    movel([0.209810, -1.227135, -2.664423, -0.820831, 1.570796, 1.780606],accel_mss,speed_ms,0,blend_radius_m)
    movel([0.209627, -1.226934, -2.664525, -0.820930, 1.570796, 1.780424],accel_mss,speed_ms,0,blend_radius_m)
    movel([0.208422, -1.226483, -2.664753, -0.821153, 1.570796, 1.779219],accel_mss,speed_ms,0,blend_radius_m)
    movel([0.205590, -1.225749, -2.665124, -0.821516, 1.570796, 1.776387],accel_mss,speed_ms,0,blend_radius_m)
    movel([0.202937, -1.225278, -2.665361, -0.821749, 1.570796, 1.773733],accel_mss,speed_ms,0,blend_radius_m)
    movel([0.200496, -1.225073, -2.665465, -0.821852, 1.570796, 1.771292],accel_mss,speed_ms,0,blend_radius_m)
    movel([0.198313, -1.225138, -2.665432, -0.821819, 1.570796, 1.769109],accel_mss,speed_ms,0,blend_radius_m)
    movel([0.196815, -1.225270, -2.665365, -0.821754, 1.570796, 1.767612],accel_mss,speed_ms,0,blend_radius_m)
    movel([0.196665, -1.225161, -2.665420, -0.821808, 1.570796, 1.767461],accel_mss,speed_ms,0,blend_radius_m)
    movel([0.196789, -1.224942, -2.665530, -0.821916, 1.570796, 1.767585],accel_mss,speed_ms,0,blend_radius_m)
    movel([0.198166, -1.223979, -2.666015, -0.822395, 1.570796, 1.768963],accel_mss,speed_ms,0,blend_radius_m)
    movel([0.198894, -1.223467, -2.666272, -0.822649, 1.570796, 1.769690],accel_mss,speed_ms,0,blend_radius_m)
    movel([0.200219, -1.222435, -2.666790, -0.823164, 1.570796, 1.771015],accel_mss,speed_ms,0,blend_radius_m)
    movel([0.200325, -1.222080, -2.666968, -0.823342, 1.570796, 1.771122],accel_mss,speed_ms,0,blend_radius_m)
    movel([0.200128, -1.221809, -2.667103, -0.823477, 1.570796, 1.770925],accel_mss,speed_ms,0,blend_radius_m)
    movel([0.199567, -1.221632, -2.667191, -0.823565, 1.570796, 1.770363],accel_mss,speed_ms,0,blend_radius_m)
    movel([0.198593, -1.221552, -2.667232, -0.823605, 1.570796, 1.769390],accel_mss,speed_ms,0,blend_radius_m)
    movel([0.196633, -1.221578, -2.667219, -0.823592, 1.570796, 1.767430],accel_mss,speed_ms,0,blend_radius_m)
    movel([0.194680, -1.221799, -2.667108, -0.823482, 1.570796, 1.765476],accel_mss,speed_ms,0,blend_radius_m)
    movel([0.192596, -1.222232, -2.666892, -0.823266, 1.570796, 1.763392],accel_mss,speed_ms,0,blend_radius_m)
    movel([0.187306, -1.223836, -2.666087, -0.822466, 1.570796, 1.758102],accel_mss,speed_ms,0,blend_radius_m)
    movel([0.188189, -1.223147, -2.666433, -0.822809, 1.570796, 1.758986],accel_mss,speed_ms,0,blend_radius_m)
    movel([0.190951, -1.221398, -2.667309, -0.823682, 1.570796, 1.761748],accel_mss,speed_ms,0,blend_radius_m)
    movel([0.191998, -1.220793, -2.667611, -0.823985, 1.570796, 1.762794],accel_mss,speed_ms,0,blend_radius_m)
    movel([0.192752, -1.220193, -2.667910, -0.824286, 1.570796, 1.763549],accel_mss,speed_ms,0,blend_radius_m)
    movel([0.192853, -1.219933, -2.668039, -0.824416, 1.570796, 1.763650],accel_mss,speed_ms,0,blend_radius_m)
    movel([0.192799, -1.219732, -2.668139, -0.824517, 1.570796, 1.763595],accel_mss,speed_ms,0,blend_radius_m)
    movel([0.192621, -1.219642, -2.668184, -0.824563, 1.570796, 1.763417],accel_mss,speed_ms,0,blend_radius_m)
    movel([0.191818, -1.219665, -2.668173, -0.824551, 1.570796, 1.762614],accel_mss,speed_ms,0,blend_radius_m)
    movel([0.190436, -1.219979, -2.668017, -0.824394, 1.570796, 1.761232],accel_mss,speed_ms,0,blend_radius_m)
    movel([0.188230, -1.220663, -2.667676, -0.824051, 1.570796, 1.759026],accel_mss,speed_ms,0,blend_radius_m)
    movel([0.185617, -1.221590, -2.667213, -0.823586, 1.570796, 1.756413],accel_mss,speed_ms,0,blend_radius_m)
    movel([0.183271, -1.222559, -2.666728, -0.823102, 1.570796, 1.754068],accel_mss,speed_ms,0,blend_radius_m)
    movel([0.181012, -1.223650, -2.666181, -0.822559, 1.570796, 1.751808],accel_mss,speed_ms,0,blend_radius_m)
    movel([0.177669, -1.225509, -2.665245, -0.821635, 1.570796, 1.748465],accel_mss,speed_ms,0,blend_radius_m)
    movel([0.176813, -1.225982, -2.665006, -0.821401, 1.570796, 1.747609],accel_mss,speed_ms,0,blend_radius_m)
    movel([0.175997, -1.226380, -2.664805, -0.821204, 1.570796, 1.746794],accel_mss,speed_ms,0,blend_radius_m)
    movel([0.178601, -1.223460, -2.666276, -0.822653, 1.570796, 1.749397],accel_mss,speed_ms,0,blend_radius_m)
    movel([0.178734, -1.223160, -2.666426, -0.822803, 1.570796, 1.749531],accel_mss,speed_ms,0,blend_radius_m)
    movel([0.178636, -1.222956, -2.666529, -0.822904, 1.570796, 1.749432],accel_mss,speed_ms,0,blend_radius_m)
    movel([0.178308, -1.222902, -2.666556, -0.822931, 1.570796, 1.749105],accel_mss,speed_ms,0,blend_radius_m)
    movel([0.177911, -1.223021, -2.666496, -0.822872, 1.570796, 1.748708],accel_mss,speed_ms,0,blend_radius_m)
    movel([0.175884, -1.224088, -2.665960, -0.822340, 1.570796, 1.746681],accel_mss,speed_ms,0,blend_radius_m)
    movel([0.172834, -1.226022, -2.664986, -0.821381, 1.570796, 1.743630],accel_mss,speed_ms,0,blend_radius_m)
    movel([0.169896, -1.228324, -2.663820, -0.820245, 1.570796, 1.740693],accel_mss,speed_ms,0,blend_radius_m)
    movel([0.167285, -1.230813, -2.662554, -0.819023, 1.570796, 1.738081],accel_mss,speed_ms,0,blend_radius_m)
    movel([0.166198, -1.232033, -2.661930, -0.818427, 1.570796, 1.736995],accel_mss,speed_ms,0,blend_radius_m)
    movel([0.164772, -1.233885, -2.660979, -0.817524, 1.570796, 1.735569],accel_mss,speed_ms,0,blend_radius_m)
    movel([0.164564, -1.234101, -2.660869, -0.817420, 1.570796, 1.735360],accel_mss,speed_ms,0,blend_radius_m)
    movel([0.164315, -1.234041, -2.660899, -0.817449, 1.570796, 1.735111],accel_mss,speed_ms,0,blend_radius_m)
    movel([0.164271, -1.233832, -2.661006, -0.817550, 1.570796, 1.735067],accel_mss,speed_ms,0,blend_radius_m)
    movel([0.164651, -1.230126, -2.662903, -0.819359, 1.570796, 1.735447],accel_mss,speed_ms,0,blend_radius_m)
    movel([0.164669, -1.229441, -2.663253, -0.819695, 1.570796, 1.735465],accel_mss,speed_ms,0,blend_radius_m)
    movel([0.164533, -1.229162, -2.663395, -0.819832, 1.570796, 1.735329],accel_mss,speed_ms,0,blend_radius_m)
    movel([0.164233, -1.229131, -2.663410, -0.819848, 1.570796, 1.735029],accel_mss,speed_ms,0,blend_radius_m)
    movel([0.163603, -1.229470, -2.663238, -0.819681, 1.570796, 1.734399],accel_mss,speed_ms,0,blend_radius_m)
    movel([0.162386, -1.230459, -2.662734, -0.819196, 1.570796, 1.733182],accel_mss,speed_ms,0,blend_radius_m)
    movel([0.159613, -1.233064, -2.661401, -0.817924, 1.570796, 1.730409],accel_mss,speed_ms,0,blend_radius_m)
    movel([0.158106, -1.234701, -2.660560, -0.817128, 1.570796, 1.728902],accel_mss,speed_ms,0,blend_radius_m)
    movel([0.156782, -1.236322, -2.659723, -0.816344, 1.570796, 1.727578],accel_mss,speed_ms,0,blend_radius_m)
    movel([0.155567, -1.238024, -2.658842, -0.815524, 1.570796, 1.726364],accel_mss,speed_ms,0,blend_radius_m)
    movel([0.154384, -1.239908, -2.657862, -0.814619, 1.570796, 1.725180],accel_mss,speed_ms,0,blend_radius_m)
    movel([0.153051, -1.242162, -2.656684, -0.813543, 1.570796, 1.723847],accel_mss,speed_ms,0,blend_radius_m)
    movel([0.152725, -1.241096, -2.657242, -0.814051, 1.570796, 1.723521],accel_mss,speed_ms,0,blend_radius_m)
    movel([0.152704, -1.240568, -2.657518, -0.814303, 1.570796, 1.723500],accel_mss,speed_ms,0,blend_radius_m)
    movel([0.153039, -1.237608, -2.659058, -0.815724, 1.570796, 1.723836],accel_mss,speed_ms,0,blend_radius_m)
    movel([0.153018, -1.237264, -2.659235, -0.815889, 1.570796, 1.723815],accel_mss,speed_ms,0,blend_radius_m)
    movel([0.152912, -1.237181, -2.659279, -0.815929, 1.570796, 1.723708],accel_mss,speed_ms,0,blend_radius_m)
    movel([0.152498, -1.237285, -2.659225, -0.815879, 1.570796, 1.723294],accel_mss,speed_ms,0,blend_radius_m)
    movel([0.152090, -1.237574, -2.659075, -0.815740, 1.570796, 1.722886],accel_mss,speed_ms,0,blend_radius_m)
    movel([0.149321, -1.240339, -2.657637, -0.814413, 1.570796, 1.720118],accel_mss,speed_ms,0,blend_radius_m)
    movel([0.146721, -1.243098, -2.656194, -0.813098, 1.570796, 1.717518],accel_mss,speed_ms,0,blend_radius_m)
    movel([0.146069, -1.243894, -2.655775, -0.812720, 1.570796, 1.716865],accel_mss,speed_ms,0,blend_radius_m)
    movel([0.144999, -1.245485, -2.654937, -0.811967, 1.570796, 1.715796],accel_mss,speed_ms,0,blend_radius_m)
    movel([0.144671, -1.245405, -2.654979, -0.812005, 1.570796, 1.715467],accel_mss,speed_ms,0,blend_radius_m)
    movel([0.144500, -1.245218, -2.655078, -0.812093, 1.570796, 1.715296],accel_mss,speed_ms,0,blend_radius_m)
    movel([0.143782, -1.244501, -2.655456, -0.812432, 1.570796, 1.714579],accel_mss,speed_ms,0,blend_radius_m)
    movel([0.143257, -1.244905, -2.655243, -0.812241, 1.570796, 1.714054],accel_mss,speed_ms,0,blend_radius_m)
    movel([0.142533, -1.246161, -2.654580, -0.811648, 1.570796, 1.713330],accel_mss,speed_ms,0,blend_radius_m)
    movel([0.141054, -1.249263, -2.652935, -0.810191, 1.570796, 1.711851],accel_mss,speed_ms,0,blend_radius_m)
    movel([0.140572, -1.250503, -2.652274, -0.809612, 1.570796, 1.711369],accel_mss,speed_ms,0,blend_radius_m)
    movel([0.140026, -1.252586, -2.651160, -0.808644, 1.570796, 1.710822],accel_mss,speed_ms,0,blend_radius_m)
    movel([0.139729, -1.254358, -2.650207, -0.807823, 1.570796, 1.710525],accel_mss,speed_ms,0,blend_radius_m)
    movel([0.139259, -1.258283, -2.648085, -0.806021, 1.570796, 1.710055],accel_mss,speed_ms,0,blend_radius_m)
    movel([0.139264, -1.259179, -2.647598, -0.805612, 1.570796, 1.710061],accel_mss,speed_ms,0,blend_radius_m)
    movel([0.138644, -1.258541, -2.647945, -0.805903, 1.570796, 1.709440],accel_mss,speed_ms,0,blend_radius_m)
    movel([0.138392, -1.258138, -2.648164, -0.806087, 1.570796, 1.709189],accel_mss,speed_ms,0,blend_radius_m)
    movel([0.137202, -1.255731, -2.649467, -0.807191, 1.570796, 1.707998],accel_mss,speed_ms,0,blend_radius_m)
    movel([0.137010, -1.255613, -2.649531, -0.807245, 1.570796, 1.707806],accel_mss,speed_ms,0,blend_radius_m)
    movel([0.136430, -1.255734, -2.649466, -0.807190, 1.570796, 1.707227],accel_mss,speed_ms,0,blend_radius_m)
    movel([0.136222, -1.255949, -2.649350, -0.807091, 1.570796, 1.707018],accel_mss,speed_ms,0,blend_radius_m)
    movel([0.136016, -1.256389, -2.649111, -0.806888, 1.570796, 1.706812],accel_mss,speed_ms,0,blend_radius_m)
    movel([0.135548, -1.257659, -2.648424, -0.806307, 1.570796, 1.706345],accel_mss,speed_ms,0,blend_radius_m)
    movel([0.135037, -1.259523, -2.647410, -0.805455, 1.570796, 1.705833],accel_mss,speed_ms,0,blend_radius_m)
    movel([0.134561, -1.262508, -2.645780, -0.804102, 1.570796, 1.705357],accel_mss,speed_ms,0,blend_radius_m)
    movel([0.134228, -1.265449, -2.644162, -0.802778, 1.570796, 1.705024],accel_mss,speed_ms,0,blend_radius_m)
    movel([0.134230, -1.267251, -2.643165, -0.801973, 1.570796, 1.705027],accel_mss,speed_ms,0,blend_radius_m)
    movel([0.134420, -1.268595, -2.642420, -0.801375, 1.570796, 1.705216],accel_mss,speed_ms,0,blend_radius_m)
    movel([0.134734, -1.270003, -2.641635, -0.800750, 1.570796, 1.705530],accel_mss,speed_ms,0,blend_radius_m)
    movel([0.135719, -1.272718, -2.640118, -0.799554, 1.570796, 1.706516],accel_mss,speed_ms,0,blend_radius_m)
    movel([0.135834, -1.273034, -2.639941, -0.799415, 1.570796, 1.706630],accel_mss,speed_ms,0,blend_radius_m)
    movel([0.135885, -1.273379, -2.639747, -0.799263, 1.570796, 1.706681],accel_mss,speed_ms,0,blend_radius_m)
    movel([0.134264, -1.273139, -2.639881, -0.799369, 1.570796, 1.705061],accel_mss,speed_ms,0,blend_radius_m)
    movel([0.133249, -1.272945, -2.639990, -0.799454, 1.570796, 1.704046],accel_mss,speed_ms,0,blend_radius_m)
    movel([0.132627, -1.272963, -2.639980, -0.799446, 1.570796, 1.703424],accel_mss,speed_ms,0,blend_radius_m)
    movel([0.132264, -1.273172, -2.639863, -0.799354, 1.570796, 1.703060],accel_mss,speed_ms,0,blend_radius_m)
    movel([0.132067, -1.273540, -2.639656, -0.799193, 1.570796, 1.702863],accel_mss,speed_ms,0,blend_radius_m)
    movel([0.132094, -1.274771, -2.638963, -0.798654, 1.570796, 1.702891],accel_mss,speed_ms,0,blend_radius_m)
    movel([0.132776, -1.277596, -2.637367, -0.797426, 1.570796, 1.703573],accel_mss,speed_ms,0,blend_radius_m)
    movel([0.133631, -1.280555, -2.635684, -0.796150, 1.570796, 1.704427],accel_mss,speed_ms,0,blend_radius_m)
    movel([0.134534, -1.283033, -2.634266, -0.795090, 1.570796, 1.705330],accel_mss,speed_ms,0,blend_radius_m)
    movel([0.135244, -1.284762, -2.633272, -0.794355, 1.570796, 1.706040],accel_mss,speed_ms,0,blend_radius_m)
    movel([0.134146, -1.285952, -2.632586, -0.793851, 1.570796, 1.704942],accel_mss,speed_ms,0,blend_radius_m)
    movel([0.133841, -1.286480, -2.632281, -0.793628, 1.570796, 1.704637],accel_mss,speed_ms,0,blend_radius_m)
    movel([0.133422, -1.287771, -2.631534, -0.793085, 1.570796, 1.704219],accel_mss,speed_ms,0,blend_radius_m)
    movel([0.133357, -1.289089, -2.630768, -0.792532, 1.570796, 1.704153],accel_mss,speed_ms,0,blend_radius_m)
    movel([0.133671, -1.290206, -2.630118, -0.792065, 1.570796, 1.704468],accel_mss,speed_ms,0,blend_radius_m)
    movel([0.134126, -1.290747, -2.629802, -0.791839, 1.570796, 1.704922],accel_mss,speed_ms,0,blend_radius_m)
    movel([0.134355, -1.290796, -2.629774, -0.791819, 1.570796, 1.705151],accel_mss,speed_ms,0,blend_radius_m)
    movel([0.134641, -1.290689, -2.629836, -0.791864, 1.570796, 1.705438],accel_mss,speed_ms,0,blend_radius_m)
    movel([0.134868, -1.290468, -2.629965, -0.791956, 1.570796, 1.705664],accel_mss,speed_ms,0,blend_radius_m)
    movel([0.134954, -1.290215, -2.630113, -0.792061, 1.570796, 1.705750],accel_mss,speed_ms,0,blend_radius_m)
    movel([0.134804, -1.289483, -2.630539, -0.792367, 1.570796, 1.705600],accel_mss,speed_ms,0,blend_radius_m)
    movel([0.134633, -1.288853, -2.630905, -0.792631, 1.570796, 1.705429],accel_mss,speed_ms,0,blend_radius_m)
    movel([0.134600, -1.288044, -2.631375, -0.792970, 1.570796, 1.705396],accel_mss,speed_ms,0,blend_radius_m)
    movel([0.134698, -1.287211, -2.631858, -0.793320, 1.570796, 1.705494],accel_mss,speed_ms,0,blend_radius_m)
    movel([0.134930, -1.286516, -2.632260, -0.793613, 1.570796, 1.705726],accel_mss,speed_ms,0,blend_radius_m)
    movel([0.135184, -1.286066, -2.632520, -0.793803, 1.570796, 1.705980],accel_mss,speed_ms,0,blend_radius_m)
    movel([0.135463, -1.285773, -2.632690, -0.793927, 1.570796, 1.706259],accel_mss,speed_ms,0,blend_radius_m)
    movel([0.135714, -1.285678, -2.632744, -0.793967, 1.570796, 1.706510],accel_mss,speed_ms,0,blend_radius_m)
    movel([0.135905, -1.285772, -2.632690, -0.793927, 1.570796, 1.706701],accel_mss,speed_ms,0,blend_radius_m)
    movel([0.136082, -1.285854, -2.632642, -0.793892, 1.570796, 1.706878],accel_mss,speed_ms,0,blend_radius_m)
    movel([0.136381, -1.285796, -2.632676, -0.793917, 1.570796, 1.707177],accel_mss,speed_ms,0,blend_radius_m)
    movel([0.136686, -1.285630, -2.632772, -0.793987, 1.570796, 1.707482],accel_mss,speed_ms,0,blend_radius_m)
    movel([0.136876, -1.285414, -2.632897, -0.794079, 1.570796, 1.707672],accel_mss,speed_ms,0,blend_radius_m)
    movel([0.136912, -1.285263, -2.632983, -0.794143, 1.570796, 1.707708],accel_mss,speed_ms,0,blend_radius_m)
    movel([0.136656, -1.284439, -2.633458, -0.794492, 1.570796, 1.707452],accel_mss,speed_ms,0,blend_radius_m)
    movel([0.135673, -1.282213, -2.634736, -0.795440, 1.570796, 1.706469],accel_mss,speed_ms,0,blend_radius_m)
    movel([0.133326, -1.274952, -2.638862, -0.798576, 1.570796, 1.704122],accel_mss,speed_ms,0,blend_radius_m)
    movel([0.133342, -1.274697, -2.639005, -0.798687, 1.570796, 1.704138],accel_mss,speed_ms,0,blend_radius_m)
    movel([0.133514, -1.274425, -2.639158, -0.798805, 1.570796, 1.704311],accel_mss,speed_ms,0,blend_radius_m)
    movel([0.135690, -1.274653, -2.639030, -0.798706, 1.570796, 1.706487],accel_mss,speed_ms,0,blend_radius_m)
    movel([0.136736, -1.274605, -2.639057, -0.798727, 1.570796, 1.707532],accel_mss,speed_ms,0,blend_radius_m)
    movel([0.137474, -1.274365, -2.639192, -0.798832, 1.570796, 1.708270],accel_mss,speed_ms,0,blend_radius_m)
    movel([0.137685, -1.274197, -2.639287, -0.798905, 1.570796, 1.708481],accel_mss,speed_ms,0,blend_radius_m)
    movel([0.137792, -1.273976, -2.639411, -0.799002, 1.570796, 1.708588],accel_mss,speed_ms,0,blend_radius_m)
    movel([0.137777, -1.273823, -2.639497, -0.799069, 1.570796, 1.708574],accel_mss,speed_ms,0,blend_radius_m)
    movel([0.137087, -1.272324, -2.640338, -0.799726, 1.570796, 1.707883],accel_mss,speed_ms,0,blend_radius_m)
    movel([0.136474, -1.270940, -2.641113, -0.800336, 1.570796, 1.707270],accel_mss,speed_ms,0,blend_radius_m)
    movel([0.135962, -1.269299, -2.642028, -0.801062, 1.570796, 1.706758],accel_mss,speed_ms,0,blend_radius_m)
    movel([0.135600, -1.267567, -2.642990, -0.801832, 1.570796, 1.706396],accel_mss,speed_ms,0,blend_radius_m)
    movel([0.135433, -1.265921, -2.643901, -0.802567, 1.570796, 1.706229],accel_mss,speed_ms,0,blend_radius_m)
    movel([0.135470, -1.264436, -2.644720, -0.803233, 1.570796, 1.706266],accel_mss,speed_ms,0,blend_radius_m)
    movel([0.135722, -1.262165, -2.645967, -0.804257, 1.570796, 1.706518],accel_mss,speed_ms,0,blend_radius_m)
    movel([0.136061, -1.259899, -2.647206, -0.805284, 1.570796, 1.706858],accel_mss,speed_ms,0,blend_radius_m)
    movel([0.136534, -1.258321, -2.648064, -0.806004, 1.570796, 1.707330],accel_mss,speed_ms,0,blend_radius_m)
    movel([0.137186, -1.258948, -2.647723, -0.805717, 1.570796, 1.707982],accel_mss,speed_ms,0,blend_radius_m)
    movel([0.137728, -1.259625, -2.647355, -0.805409, 1.570796, 1.708524],accel_mss,speed_ms,0,blend_radius_m)
    movel([0.139104, -1.260707, -2.646765, -0.804917, 1.570796, 1.709901],accel_mss,speed_ms,0,blend_radius_m)
    movel([0.139721, -1.260930, -2.646643, -0.804816, 1.570796, 1.710517],accel_mss,speed_ms,0,blend_radius_m)
    movel([0.140174, -1.260939, -2.646638, -0.804812, 1.570796, 1.710970],accel_mss,speed_ms,0,blend_radius_m)
    movel([0.140323, -1.260838, -2.646693, -0.804858, 1.570796, 1.711119],accel_mss,speed_ms,0,blend_radius_m)
    movel([0.140648, -1.260367, -2.646951, -0.805072, 1.570796, 1.711444],accel_mss,speed_ms,0,blend_radius_m)
    movel([0.140708, -1.260067, -2.647114, -0.805208, 1.570796, 1.711504],accel_mss,speed_ms,0,blend_radius_m)
    movel([0.140526, -1.258193, -2.648134, -0.806062, 1.570796, 1.711323],accel_mss,speed_ms,0,blend_radius_m)
    movel([0.140540, -1.257336, -2.648599, -0.806454, 1.570796, 1.711337],accel_mss,speed_ms,0,blend_radius_m)
    movel([0.140917, -1.254345, -2.650214, -0.807829, 1.570796, 1.711714],accel_mss,speed_ms,0,blend_radius_m)
    movel([0.141310, -1.252044, -2.651450, -0.808895, 1.570796, 1.712106],accel_mss,speed_ms,0,blend_radius_m)
    movel([0.141704, -1.250443, -2.652306, -0.809640, 1.570796, 1.712500],accel_mss,speed_ms,0,blend_radius_m)
    movel([0.142246, -1.248970, -2.653091, -0.810329, 1.570796, 1.713042],accel_mss,speed_ms,0,blend_radius_m)
    movel([0.143090, -1.247163, -2.654050, -0.811176, 1.570796, 1.713886],accel_mss,speed_ms,0,blend_radius_m)
    movel([0.143399, -1.246554, -2.654372, -0.811463, 1.570796, 1.714195],accel_mss,speed_ms,0,blend_radius_m)
    movel([0.144020, -1.246823, -2.654230, -0.811336, 1.570796, 1.714816],accel_mss,speed_ms,0,blend_radius_m)
    movel([0.144282, -1.246919, -2.654179, -0.811291, 1.570796, 1.715078],accel_mss,speed_ms,0,blend_radius_m)
    movel([0.144972, -1.246990, -2.654142, -0.811258, 1.570796, 1.715768],accel_mss,speed_ms,0,blend_radius_m)
    movel([0.145157, -1.246868, -2.654206, -0.811315, 1.570796, 1.715954],accel_mss,speed_ms,0,blend_radius_m)
    movel([0.146182, -1.245466, -2.654947, -0.811976, 1.570796, 1.716978],accel_mss,speed_ms,0,blend_radius_m)
    movel([0.147089, -1.244204, -2.655612, -0.812573, 1.570796, 1.717885],accel_mss,speed_ms,0,blend_radius_m)
    movel([0.148829, -1.242153, -2.656689, -0.813547, 1.570796, 1.719625],accel_mss,speed_ms,0,blend_radius_m)
    movel([0.150689, -1.240056, -2.657785, -0.814548, 1.570796, 1.721485],accel_mss,speed_ms,0,blend_radius_m)
    movel([0.151224, -1.239699, -2.657971, -0.814719, 1.570796, 1.722020],accel_mss,speed_ms,0,blend_radius_m)
    movel([0.151439, -1.240876, -2.657357, -0.814156, 1.570796, 1.722236],accel_mss,speed_ms,0,blend_radius_m)
    movel([0.151574, -1.241880, -2.656832, -0.813677, 1.570796, 1.722371],accel_mss,speed_ms,0,blend_radius_m)
    movel([0.151908, -1.242903, -2.656296, -0.813190, 1.570796, 1.722705],accel_mss,speed_ms,0,blend_radius_m)
    movel([0.152333, -1.243743, -2.655855, -0.812791, 1.570796, 1.723129],accel_mss,speed_ms,0,blend_radius_m)
    movel([0.152747, -1.244020, -2.655709, -0.812660, 1.570796, 1.723544],accel_mss,speed_ms,0,blend_radius_m)
    movel([0.153064, -1.243966, -2.655738, -0.812686, 1.570796, 1.723860],accel_mss,speed_ms,0,blend_radius_m)
    movel([0.153430, -1.243719, -2.655867, -0.812803, 1.570796, 1.724226],accel_mss,speed_ms,0,blend_radius_m)
    movel([0.153740, -1.243358, -2.656057, -0.812974, 1.570796, 1.724536],accel_mss,speed_ms,0,blend_radius_m)
    movel([0.153890, -1.242987, -2.656251, -0.813150, 1.570796, 1.724687],accel_mss,speed_ms,0,blend_radius_m)
    movel([0.154111, -1.242366, -2.656577, -0.813446, 1.570796, 1.724907],accel_mss,speed_ms,0,blend_radius_m)
    movel([0.154958, -1.240833, -2.657379, -0.814177, 1.570796, 1.725754],accel_mss,speed_ms,0,blend_radius_m)
    movel([0.155913, -1.239224, -2.658218, -0.814947, 1.570796, 1.726710],accel_mss,speed_ms,0,blend_radius_m)
    movel([0.157932, -1.236373, -2.659697, -0.816319, 1.570796, 1.728728],accel_mss,speed_ms,0,blend_radius_m)
    movel([0.159064, -1.235000, -2.660405, -0.816983, 1.570796, 1.729860],accel_mss,speed_ms,0,blend_radius_m)
    movel([0.161569, -1.232437, -2.661723, -0.818229, 1.570796, 1.732365],accel_mss,speed_ms,0,blend_radius_m)
    movel([0.163243, -1.230891, -2.662513, -0.818985, 1.570796, 1.734040],accel_mss,speed_ms,0,blend_radius_m)
    movel([0.163144, -1.231742, -2.662079, -0.818569, 1.570796, 1.733940],accel_mss,speed_ms,0,blend_radius_m)
    movel([0.163031, -1.233719, -2.661065, -0.817605, 1.570796, 1.733827],accel_mss,speed_ms,0,blend_radius_m)
    movel([0.163214, -1.235199, -2.660303, -0.816887, 1.570796, 1.734010],accel_mss,speed_ms,0,blend_radius_m)
    movel([0.163648, -1.236087, -2.659845, -0.816457, 1.570796, 1.734445],accel_mss,speed_ms,0,blend_radius_m)
    movel([0.163922, -1.236243, -2.659764, -0.816382, 1.570796, 1.734718],accel_mss,speed_ms,0,blend_radius_m)
    movel([0.164312, -1.236210, -2.659781, -0.816398, 1.570796, 1.735108],accel_mss,speed_ms,0,blend_radius_m)
    movel([0.165194, -1.234980, -2.660416, -0.816993, 1.570796, 1.735990],accel_mss,speed_ms,0,blend_radius_m)
    movel([0.166079, -1.233746, -2.661051, -0.817592, 1.570796, 1.736875],accel_mss,speed_ms,0,blend_radius_m)
    movel([0.168287, -1.231150, -2.662381, -0.818858, 1.570796, 1.739083],accel_mss,speed_ms,0,blend_radius_m)
    movel([0.169460, -1.229964, -2.662986, -0.819439, 1.570796, 1.740256],accel_mss,speed_ms,0,blend_radius_m)
    movel([0.172229, -1.227653, -2.664161, -0.820575, 1.570796, 1.743025],accel_mss,speed_ms,0,blend_radius_m)
    movel([0.173842, -1.226444, -2.664772, -0.821172, 1.570796, 1.744638],accel_mss,speed_ms,0,blend_radius_m)
    movel([0.174837, -1.225808, -2.665094, -0.821487, 1.570796, 1.745633],accel_mss,speed_ms,0,blend_radius_m)
    movel([0.175334, -1.225534, -2.665232, -0.821623, 1.570796, 1.746131],accel_mss,speed_ms,0,blend_radius_m)
    movel([0.174097, -1.227664, -2.664155, -0.820570, 1.570796, 1.744893],accel_mss,speed_ms,0,blend_radius_m)
    movel([0.173869, -1.228208, -2.663879, -0.820302, 1.570796, 1.744666],accel_mss,speed_ms,0,blend_radius_m)
    movel([0.173848, -1.228549, -2.663706, -0.820134, 1.570796, 1.744644],accel_mss,speed_ms,0,blend_radius_m)
    movel([0.174006, -1.228765, -2.663597, -0.820028, 1.570796, 1.744802],accel_mss,speed_ms,0,blend_radius_m)
    movel([0.174215, -1.228770, -2.663594, -0.820025, 1.570796, 1.745011],accel_mss,speed_ms,0,blend_radius_m)
    movel([0.174561, -1.228627, -2.663666, -0.820095, 1.570796, 1.745357],accel_mss,speed_ms,0,blend_radius_m)
    movel([0.175949, -1.227750, -2.664112, -0.820528, 1.570796, 1.746745],accel_mss,speed_ms,0,blend_radius_m)
    movel([0.177628, -1.226651, -2.664668, -0.821070, 1.570796, 1.748424],accel_mss,speed_ms,0,blend_radius_m)
    movel([0.180743, -1.224882, -2.665561, -0.821946, 1.570796, 1.751539],accel_mss,speed_ms,0,blend_radius_m)
    movel([0.182561, -1.223995, -2.666007, -0.822387, 1.570796, 1.753358],accel_mss,speed_ms,0,blend_radius_m)
    movel([0.186299, -1.222416, -2.666799, -0.823174, 1.570796, 1.757095],accel_mss,speed_ms,0,blend_radius_m)
    movel([0.188195, -1.221690, -2.667163, -0.823536, 1.570796, 1.758992],accel_mss,speed_ms,0,blend_radius_m)
    movel([0.188266, -1.221843, -2.667086, -0.823460, 1.570796, 1.759062],accel_mss,speed_ms,0,blend_radius_m)
    movel([0.187893, -1.222163, -2.666926, -0.823300, 1.570796, 1.758689],accel_mss,speed_ms,0,blend_radius_m)
    movel([0.184761, -1.224830, -2.665587, -0.821972, 1.570796, 1.755557],accel_mss,speed_ms,0,blend_radius_m)
    movel([0.183850, -1.225731, -2.665133, -0.821525, 1.570796, 1.754646],accel_mss,speed_ms,0,blend_radius_m)
    movel([0.183653, -1.226162, -2.664915, -0.821312, 1.570796, 1.754450],accel_mss,speed_ms,0,blend_radius_m)
    movel([0.184058, -1.226438, -2.664776, -0.821175, 1.570796, 1.754854],accel_mss,speed_ms,0,blend_radius_m)
    movel([0.184382, -1.226354, -2.664818, -0.821217, 1.570796, 1.755179],accel_mss,speed_ms,0,blend_radius_m)
    movel([0.186555, -1.225356, -2.665322, -0.821711, 1.570796, 1.757351],accel_mss,speed_ms,0,blend_radius_m)
    movel([0.187622, -1.224945, -2.665529, -0.821915, 1.570796, 1.758418],accel_mss,speed_ms,0,blend_radius_m)
    movel([0.192817, -1.223378, -2.666317, -0.822694, 1.570796, 1.763614],accel_mss,speed_ms,0,blend_radius_m)
    movel([0.194080, -1.223078, -2.666467, -0.822843, 1.570796, 1.764876],accel_mss,speed_ms,0,blend_radius_m)
    movel([0.196968, -1.222803, -2.666606, -0.822981, 1.570796, 1.767764],accel_mss,speed_ms,0,blend_radius_m)
    movel([0.197569, -1.222793, -2.666611, -0.822986, 1.570796, 1.768365],accel_mss,speed_ms,0,blend_radius_m)
    movel([0.198106, -1.222817, -2.666599, -0.822974, 1.570796, 1.768902],accel_mss,speed_ms,0,blend_radius_m)
    movel([0.195737, -1.224537, -2.665734, -0.822117, 1.570796, 1.766533],accel_mss,speed_ms,0,blend_radius_m)
    movel([0.194465, -1.225446, -2.665276, -0.821666, 1.570796, 1.765261],accel_mss,speed_ms,0,blend_radius_m)
    movel([0.193490, -1.226305, -2.664843, -0.821241, 1.570796, 1.764286],accel_mss,speed_ms,0,blend_radius_m)
    movel([0.193369, -1.226594, -2.664697, -0.821098, 1.570796, 1.764165],accel_mss,speed_ms,0,blend_radius_m)
    movel([0.193412, -1.226791, -2.664597, -0.821001, 1.570796, 1.764208],accel_mss,speed_ms,0,blend_radius_m)
    movel([0.193565, -1.226888, -2.664548, -0.820953, 1.570796, 1.764361],accel_mss,speed_ms,0,blend_radius_m)
    movel([0.194478, -1.226815, -2.664585, -0.820989, 1.570796, 1.765274],accel_mss,speed_ms,0,blend_radius_m)
    movel([0.196240, -1.226553, -2.664718, -0.821118, 1.570796, 1.767037],accel_mss,speed_ms,0,blend_radius_m)
    movel([0.198966, -1.226322, -2.664835, -0.821233, 1.570796, 1.769762],accel_mss,speed_ms,0,blend_radius_m)
    movel([0.200218, -1.226326, -2.664833, -0.821231, 1.570796, 1.771015],accel_mss,speed_ms,0,blend_radius_m)
    movel([0.204234, -1.226849, -2.664568, -0.820972, 1.570796, 1.775030],accel_mss,speed_ms,0,blend_radius_m)
    movel([0.206740, -1.227318, -2.664331, -0.820741, 1.570796, 1.777536],accel_mss,speed_ms,0,blend_radius_m)
    movel([0.206852, -1.227516, -2.664230, -0.820643, 1.570796, 1.777648],accel_mss,speed_ms,0,blend_radius_m)
    movel([0.204924, -1.228736, -2.663611, -0.820042, 1.570796, 1.775720],accel_mss,speed_ms,0,blend_radius_m)
    movel([0.203880, -1.229532, -2.663206, -0.819651, 1.570796, 1.774677],accel_mss,speed_ms,0,blend_radius_m)
    movel([0.203054, -1.230302, -2.662814, -0.819273, 1.570796, 1.773851],accel_mss,speed_ms,0,blend_radius_m)
    movel([0.202816, -1.230764, -2.662578, -0.819047, 1.570796, 1.773613],accel_mss,speed_ms,0,blend_radius_m)
    movel([0.202895, -1.230964, -2.662476, -0.818949, 1.570796, 1.773691],accel_mss,speed_ms,0,blend_radius_m)
    movel([0.203150, -1.231040, -2.662438, -0.818912, 1.570796, 1.773946],accel_mss,speed_ms,0,blend_radius_m)
    movel([0.204940, -1.230824, -2.662547, -0.819017, 1.570796, 1.775736],accel_mss,speed_ms,0,blend_radius_m)
    movel([0.207699, -1.230528, -2.662699, -0.819162, 1.570796, 1.778496],accel_mss,speed_ms,0,blend_radius_m)
    movel([0.210248, -1.230533, -2.662696, -0.819160, 1.570796, 1.781044],accel_mss,speed_ms,0,blend_radius_m)
    movel([0.212928, -1.230861, -2.662529, -0.818999, 1.570796, 1.783724],accel_mss,speed_ms,0,blend_radius_m)
    movel([0.216125, -1.231553, -2.662175, -0.818661, 1.570796, 1.786921],accel_mss,speed_ms,0,blend_radius_m)
    movel([0.218727, -1.232216, -2.661836, -0.818337, 1.570796, 1.789523],accel_mss,speed_ms,0,blend_radius_m)
    movel([0.216739, -1.232863, -2.661504, -0.818022, 1.570796, 1.787536],accel_mss,speed_ms,0,blend_radius_m)
    movel([0.214968, -1.233496, -2.661180, -0.817714, 1.570796, 1.785765],accel_mss,speed_ms,0,blend_radius_m)
    movel([0.214624, -1.233691, -2.661079, -0.817619, 1.570796, 1.785420],accel_mss,speed_ms,0,blend_radius_m)
    movel([0.214327, -1.233979, -2.660931, -0.817479, 1.570796, 1.785124],accel_mss,speed_ms,0,blend_radius_m)
    movel([0.214208, -1.234240, -2.660797, -0.817352, 1.570796, 1.785004],accel_mss,speed_ms,0,blend_radius_m)
    movel([0.214277, -1.234433, -2.660698, -0.817259, 1.570796, 1.785073],accel_mss,speed_ms,0,blend_radius_m)
    movel([0.216667, -1.235597, -2.660098, -0.816694, 1.570796, 1.787463],accel_mss,speed_ms,0,blend_radius_m)
    movel([0.219523, -1.236952, -2.659397, -0.816040, 1.570796, 1.790319],accel_mss,speed_ms,0,blend_radius_m)
    movel([0.222909, -1.238643, -2.658520, -0.815226, 1.570796, 1.793705],accel_mss,speed_ms,0,blend_radius_m)
    movel([0.222907, -1.238777, -2.658451, -0.815162, 1.570796, 1.793704],accel_mss,speed_ms,0,blend_radius_m)
    movel([0.222102, -1.239021, -2.658324, -0.815044, 1.570796, 1.792898],accel_mss,speed_ms,0,blend_radius_m)
    movel([0.221775, -1.239273, -2.658192, -0.814923, 1.570796, 1.792571],accel_mss,speed_ms,0,blend_radius_m)
    movel([0.221635, -1.239497, -2.658076, -0.814816, 1.570796, 1.792431],accel_mss,speed_ms,0,blend_radius_m)
    movel([0.221663, -1.239820, -2.657908, -0.814661, 1.570796, 1.792459],accel_mss,speed_ms,0,blend_radius_m)
    movel([0.222321, -1.240976, -2.657305, -0.814108, 1.570796, 1.793117],accel_mss,speed_ms,0,blend_radius_m)
    movel([0.223076, -1.242193, -2.656668, -0.813528, 1.570796, 1.793872],accel_mss,speed_ms,0,blend_radius_m)
    movel([0.224791, -1.244435, -2.655490, -0.812463, 1.570796, 1.795587],accel_mss,speed_ms,0,blend_radius_m)
    movel([0.226110, -1.245787, -2.654778, -0.811824, 1.570796, 1.796907],accel_mss,speed_ms,0,blend_radius_m)
    movel([0.229227, -1.248487, -2.653348, -0.810555, 1.570796, 1.800024],accel_mss,speed_ms,0,blend_radius_m)
    movel([0.227819, -1.247990, -2.653611, -0.810787, 1.570796, 1.798616],accel_mss,speed_ms,0,blend_radius_m)
    movel([0.227199, -1.247705, -2.653763, -0.810922, 1.570796, 1.797996],accel_mss,speed_ms,0,blend_radius_m)
    movel([0.226711, -1.247667, -2.653783, -0.810939, 1.570796, 1.797507],accel_mss,speed_ms,0,blend_radius_m)
    movel([0.226373, -1.247858, -2.653681, -0.810850, 1.570796, 1.797170],accel_mss,speed_ms,0,blend_radius_m)
    movel([0.226162, -1.248222, -2.653488, -0.810679, 1.570796, 1.796958],accel_mss,speed_ms,0,blend_radius_m)
    movel([0.226191, -1.248619, -2.653277, -0.810493, 1.570796, 1.796987],accel_mss,speed_ms,0,blend_radius_m)
    movel([0.228277, -1.252344, -2.651289, -0.808756, 1.570796, 1.799073],accel_mss,speed_ms,0,blend_radius_m)
    movel([0.229256, -1.253853, -2.650479, -0.808057, 1.570796, 1.800052],accel_mss,speed_ms,0,blend_radius_m)
    movel([0.231055, -1.256094, -2.649271, -0.807024, 1.570796, 1.801851],accel_mss,speed_ms,0,blend_radius_m)
    movel([0.232001, -1.257075, -2.648740, -0.806574, 1.570796, 1.802797],accel_mss,speed_ms,0,blend_radius_m)
    movel([0.233728, -1.258544, -2.647943, -0.805902, 1.570796, 1.804525],accel_mss,speed_ms,0,blend_radius_m)
    movel([0.232321, -1.258288, -2.648082, -0.806019, 1.570796, 1.803118],accel_mss,speed_ms,0,blend_radius_m)
    movel([0.231902, -1.258344, -2.648052, -0.805993, 1.570796, 1.802698],accel_mss,speed_ms,0,blend_radius_m)
    movel([0.231611, -1.258549, -2.647941, -0.805900, 1.570796, 1.802407],accel_mss,speed_ms,0,blend_radius_m)
    movel([0.231434, -1.258876, -2.647763, -0.805750, 1.570796, 1.802231],accel_mss,speed_ms,0,blend_radius_m)
    movel([0.231668, -1.259671, -2.647330, -0.805388, 1.570796, 1.802464],accel_mss,speed_ms,0,blend_radius_m)
    movel([0.231970, -1.260348, -2.646961, -0.805080, 1.570796, 1.802766],accel_mss,speed_ms,0,blend_radius_m)
    movel([0.234476, -1.264568, -2.644647, -0.803173, 1.570796, 1.805273],accel_mss,speed_ms,0,blend_radius_m)
    movel([0.235504, -1.265899, -2.643913, -0.802577, 1.570796, 1.806300],accel_mss,speed_ms,0,blend_radius_m)
    movel([0.236658, -1.267116, -2.643240, -0.802033, 1.570796, 1.807454],accel_mss,speed_ms,0,blend_radius_m)
    movel([0.237777, -1.268067, -2.642713, -0.801609, 1.570796, 1.808573],accel_mss,speed_ms,0,blend_radius_m)
    movel([0.239018, -1.268891, -2.642255, -0.801243, 1.570796, 1.809814],accel_mss,speed_ms,0,blend_radius_m)
    movel([0.240296, -1.269527, -2.641901, -0.800961, 1.570796, 1.811093],accel_mss,speed_ms,0,blend_radius_m)
    movel([0.241693, -1.270013, -2.641630, -0.800746, 1.570796, 1.812489],accel_mss,speed_ms,0,blend_radius_m)
    movel([0.243358, -1.270481, -2.641369, -0.800539, 1.570796, 1.814154],accel_mss,speed_ms,0,blend_radius_m)
    movel([0.242221, -1.270780, -2.641202, -0.800407, 1.570796, 1.813017],accel_mss,speed_ms,0,blend_radius_m)
    movel([0.241651, -1.270900, -2.641135, -0.800354, 1.570796, 1.812448],accel_mss,speed_ms,0,blend_radius_m)
    movel([0.239946, -1.270947, -2.641109, -0.800333, 1.570796, 1.810742],accel_mss,speed_ms,0,blend_radius_m)
    movel([0.239120, -1.270885, -2.641144, -0.800361, 1.570796, 1.809917],accel_mss,speed_ms,0,blend_radius_m)
    movel([0.238617, -1.270959, -2.641102, -0.800328, 1.570796, 1.809414],accel_mss,speed_ms,0,blend_radius_m)
    movel([0.238307, -1.271167, -2.640986, -0.800236, 1.570796, 1.809103],accel_mss,speed_ms,0,blend_radius_m)
    movel([0.238115, -1.271508, -2.640795, -0.800086, 1.570796, 1.808911],accel_mss,speed_ms,0,blend_radius_m)
    movel([0.238209, -1.271964, -2.640540, -0.799885, 1.570796, 1.809005],accel_mss,speed_ms,0,blend_radius_m)
    movel([0.239383, -1.273036, -2.639939, -0.799414, 1.570796, 1.810179],accel_mss,speed_ms,0,blend_radius_m)
    movel([0.240763, -1.274126, -2.639327, -0.798936, 1.570796, 1.811560],accel_mss,speed_ms,0,blend_radius_m)
    movel([0.242193, -1.275048, -2.638807, -0.798533, 1.570796, 1.812990],accel_mss,speed_ms,0,blend_radius_m)
    movel([0.243693, -1.275781, -2.638394, -0.798214, 1.570796, 1.814489],accel_mss,speed_ms,0,blend_radius_m)
    movel([0.245668, -1.276513, -2.637980, -0.797896, 1.570796, 1.816464],accel_mss,speed_ms,0,blend_radius_m)
    movel([0.247673, -1.277113, -2.637641, -0.797635, 1.570796, 1.818470],accel_mss,speed_ms,0,blend_radius_m)
    movel([0.249757, -1.277474, -2.637436, -0.797479, 1.570796, 1.820553],accel_mss,speed_ms,0,blend_radius_m)
    movel([0.250172, -1.277551, -2.637392, -0.797445, 1.570796, 1.820968],accel_mss,speed_ms,0,blend_radius_m)
    movel([0.250531, -1.277690, -2.637314, -0.797385, 1.570796, 1.821327],accel_mss,speed_ms,0,blend_radius_m)
    movel([0.250404, -1.277843, -2.637227, -0.797319, 1.570796, 1.821200],accel_mss,speed_ms,0,blend_radius_m)
    movel([0.247937, -1.279052, -2.636540, -0.796797, 1.570796, 1.818733],accel_mss,speed_ms,0,blend_radius_m)
    movel([0.247569, -1.279222, -2.636443, -0.796723, 1.570796, 1.818365],accel_mss,speed_ms,0,blend_radius_m)
    movel([0.247188, -1.279552, -2.636256, -0.796581, 1.570796, 1.817984],accel_mss,speed_ms,0,blend_radius_m)
    movel([0.247094, -1.279767, -2.636133, -0.796489, 1.570796, 1.817891],accel_mss,speed_ms,0,blend_radius_m)
    movel([0.247095, -1.280267, -2.635848, -0.796274, 1.570796, 1.817892],accel_mss,speed_ms,0,blend_radius_m)
    movel([0.247377, -1.280586, -2.635666, -0.796137, 1.570796, 1.818174],accel_mss,speed_ms,0,blend_radius_m)
    movel([0.250234, -1.281902, -2.634914, -0.795573, 1.570796, 1.821030],accel_mss,speed_ms,0,blend_radius_m)
    movel([0.253359, -1.283041, -2.634262, -0.795087, 1.570796, 1.824155],accel_mss,speed_ms,0,blend_radius_m)
    movel([0.256069, -1.283598, -2.633942, -0.794849, 1.570796, 1.826866],accel_mss,speed_ms,0,blend_radius_m)
    movel([0.257177, -1.283747, -2.633856, -0.794786, 1.570796, 1.827973],accel_mss,speed_ms,0,blend_radius_m)
    movel([0.257323, -1.283919, -2.633757, -0.794713, 1.570796, 1.828120],accel_mss,speed_ms,0,blend_radius_m)
    movel([0.257153, -1.284125, -2.633639, -0.794625, 1.570796, 1.827949],accel_mss,speed_ms,0,blend_radius_m)
    movel([0.256066, -1.284490, -2.633429, -0.794470, 1.570796, 1.826862],accel_mss,speed_ms,0,blend_radius_m)
    movel([0.254886, -1.284953, -2.633162, -0.794274, 1.570796, 1.825682],accel_mss,speed_ms,0,blend_radius_m)
    movel([0.254606, -1.285153, -2.633047, -0.794189, 1.570796, 1.825403],accel_mss,speed_ms,0,blend_radius_m)
    movel([0.254428, -1.285428, -2.632889, -0.794073, 1.570796, 1.825225],accel_mss,speed_ms,0,blend_radius_m)
    movel([0.254409, -1.285681, -2.632742, -0.793966, 1.570796, 1.825205],accel_mss,speed_ms,0,blend_radius_m)
    movel([0.254553, -1.285833, -2.632655, -0.793901, 1.570796, 1.825349],accel_mss,speed_ms,0,blend_radius_m)
    movel([0.256091, -1.286069, -2.632518, -0.793801, 1.570796, 1.826887],accel_mss,speed_ms,0,blend_radius_m)
    movel([0.256821, -1.286022, -2.632546, -0.793821, 1.570796, 1.827617],accel_mss,speed_ms,0,blend_radius_m)
    movel([0.260543, -1.285348, -2.632934, -0.794106, 1.570796, 1.831339],accel_mss,speed_ms,0,blend_radius_m)
    movel([0.261452, -1.285104, -2.633075, -0.794210, 1.570796, 1.832248],accel_mss,speed_ms,0,blend_radius_m)
    movel([0.264193, -1.283903, -2.633767, -0.794720, 1.570796, 1.834989],accel_mss,speed_ms,0,blend_radius_m)
    movel([0.264822, -1.283621, -2.633929, -0.794839, 1.570796, 1.835618],accel_mss,speed_ms,0,blend_radius_m)
    movel([0.265426, -1.283394, -2.634059, -0.794936, 1.570796, 1.836222],accel_mss,speed_ms,0,blend_radius_m)
    movel([0.264918, -1.284397, -2.633482, -0.794510, 1.570796, 1.835714],accel_mss,speed_ms,0,blend_radius_m)
    movel([0.264262, -1.285608, -2.632785, -0.793997, 1.570796, 1.835059],accel_mss,speed_ms,0,blend_radius_m)
    movel([0.264214, -1.285844, -2.632648, -0.793897, 1.570796, 1.835010],accel_mss,speed_ms,0,blend_radius_m)
    movel([0.264316, -1.286004, -2.632556, -0.793829, 1.570796, 1.835112],accel_mss,speed_ms,0,blend_radius_m)
    movel([0.264532, -1.286040, -2.632535, -0.793814, 1.570796, 1.835328],accel_mss,speed_ms,0,blend_radius_m)
    movel([0.264796, -1.285934, -2.632596, -0.793859, 1.570796, 1.835593],accel_mss,speed_ms,0,blend_radius_m)
    movel([0.266034, -1.285075, -2.633092, -0.794222, 1.570796, 1.836830],accel_mss,speed_ms,0,blend_radius_m)
    movel([0.267531, -1.283887, -2.633775, -0.794726, 1.570796, 1.838327],accel_mss,speed_ms,0,blend_radius_m)
    movel([0.268962, -1.282609, -2.634509, -0.795271, 1.570796, 1.839758],accel_mss,speed_ms,0,blend_radius_m)
    movel([0.272019, -1.279479, -2.636297, -0.796613, 1.570796, 1.842816],accel_mss,speed_ms,0,blend_radius_m)
    movel([0.274765, -1.276177, -2.638170, -0.798042, 1.570796, 1.845561],accel_mss,speed_ms,0,blend_radius_m)
    movel([0.275814, -1.274708, -2.638999, -0.798682, 1.570796, 1.846610],accel_mss,speed_ms,0,blend_radius_m)
    movel([0.276737, -1.273204, -2.639845, -0.799340, 1.570796, 1.847533],accel_mss,speed_ms,0,blend_radius_m)
    movel([0.276930, -1.272872, -2.640031, -0.799486, 1.570796, 1.847727],accel_mss,speed_ms,0,blend_radius_m)
    movel([0.277357, -1.272321, -2.640340, -0.799728, 1.570796, 1.848154],accel_mss,speed_ms,0,blend_radius_m)
    movel([0.277788, -1.273329, -2.639775, -0.799285, 1.570796, 1.848585],accel_mss,speed_ms,0,blend_radius_m)
    movel([0.278170, -1.274254, -2.639255, -0.798880, 1.570796, 1.848966],accel_mss,speed_ms,0,blend_radius_m)
    movel([0.278353, -1.274337, -2.639208, -0.798844, 1.570796, 1.849150],accel_mss,speed_ms,0,blend_radius_m)
    movel([0.278618, -1.274224, -2.639272, -0.798894, 1.570796, 1.849414],accel_mss,speed_ms,0,blend_radius_m)
    movel([0.278939, -1.273911, -2.639448, -0.799030, 1.570796, 1.849735],accel_mss,speed_ms,0,blend_radius_m)
    movel([0.279169, -1.273553, -2.639649, -0.799187, 1.570796, 1.849966],accel_mss,speed_ms,0,blend_radius_m)
    movel([0.280084, -1.271532, -2.640782, -0.800075, 1.570796, 1.850880],accel_mss,speed_ms,0,blend_radius_m)
    movel([0.281671, -1.267472, -2.643043, -0.801874, 1.570796, 1.852468],accel_mss,speed_ms,0,blend_radius_m)
    movel([0.282759, -1.263869, -2.645032, -0.803488, 1.570796, 1.853555],accel_mss,speed_ms,0,blend_radius_m)
    movel([0.283457, -1.260288, -2.646993, -0.805107, 1.570796, 1.854254],accel_mss,speed_ms,0,blend_radius_m)
    movel([0.283890, -1.256132, -2.649250, -0.807007, 1.570796, 1.854686],accel_mss,speed_ms,0,blend_radius_m)
    movel([0.284536, -1.257773, -2.648362, -0.806254, 1.570796, 1.855332],accel_mss,speed_ms,0,blend_radius_m)
    movel([0.284743, -1.257841, -2.648325, -0.806223, 1.570796, 1.855539],accel_mss,speed_ms,0,blend_radius_m)
    movel([0.285051, -1.257727, -2.648387, -0.806275, 1.570796, 1.855847],accel_mss,speed_ms,0,blend_radius_m)
    movel([0.285376, -1.257416, -2.648555, -0.806417, 1.570796, 1.856173],accel_mss,speed_ms,0,blend_radius_m)
    movel([0.285614, -1.256958, -2.648804, -0.806628, 1.570796, 1.856410],accel_mss,speed_ms,0,blend_radius_m)
    movel([0.285837, -1.256166, -2.649232, -0.806991, 1.570796, 1.856634],accel_mss,speed_ms,0,blend_radius_m)
    movel([0.286065, -1.255050, -2.649835, -0.807504, 1.570796, 1.856862],accel_mss,speed_ms,0,blend_radius_m)
    speed_ms = 0.005
    movel([0.286065, -1.245601, -2.645271, -0.821517, 1.570796, 1.856862],accel_mss,speed_ms,0,blend_radius_m)
    speed_ms = 0.040
    movel([0.268123, -1.229245, -2.653817, -0.829327, 1.570796, 1.838920],accel_mss,speed_ms,0,blend_radius_m)
    speed_ms = 0.005
    movel([0.268123, -1.238768, -2.658455, -0.815166, 1.570796, 1.838920],accel_mss,speed_ms,0,blend_radius_m)
    speed_ms = 0.025
    movel([0.268330, -1.240278, -2.657669, -0.814442, 1.570796, 1.839126],accel_mss,speed_ms,0,blend_radius_m)
    movel([0.267669, -1.239958, -2.657836, -0.814595, 1.570796, 1.838465],accel_mss,speed_ms,0,blend_radius_m)
    movel([0.267290, -1.239606, -2.658019, -0.814764, 1.570796, 1.838086],accel_mss,speed_ms,0,blend_radius_m)
    movel([0.267172, -1.239273, -2.658193, -0.814924, 1.570796, 1.837968],accel_mss,speed_ms,0,blend_radius_m)
    movel([0.267257, -1.238823, -2.658427, -0.815139, 1.570796, 1.838053],accel_mss,speed_ms,0,blend_radius_m)
    movel([0.267776, -1.237740, -2.658989, -0.815660, 1.570796, 1.838572],accel_mss,speed_ms,0,blend_radius_m)
    movel([0.268123, -1.238768, -2.658455, -0.815166, 1.570796, 1.838920],accel_mss,speed_ms,0,blend_radius_m)
    movel([0.268330, -1.240278, -2.657669, -0.814442, 1.570796, 1.839126],accel_mss,speed_ms,0,blend_radius_m)
    movel([0.267669, -1.239958, -2.657836, -0.814595, 1.570796, 1.838465],accel_mss,speed_ms,0,blend_radius_m)
    speed_ms = 0.005
    movel([0.267669, -1.230439, -2.653204, -0.828746, 1.570796, 1.838465],accel_mss,speed_ms,0,blend_radius_m)
    speed_ms = 0.040
    movel([0.271645, -1.189183, -2.673465, -0.849741, 1.570796, 1.842441],accel_mss,speed_ms,0,blend_radius_m)
    speed_ms = 0.005
    movel([0.271645, -1.198861, -2.678284, -0.835244, 1.570796, 1.842441],accel_mss,speed_ms,0,blend_radius_m)
    speed_ms = 0.025
    movel([0.272020, -1.198260, -2.678569, -0.835560, 1.570796, 1.842817],accel_mss,speed_ms,0,blend_radius_m)
    movel([0.272063, -1.197955, -2.678713, -0.835721, 1.570796, 1.842860],accel_mss,speed_ms,0,blend_radius_m)
    movel([0.271607, -1.197834, -2.678770, -0.835784, 1.570796, 1.842404],accel_mss,speed_ms,0,blend_radius_m)
    movel([0.271155, -1.197426, -2.678964, -0.835999, 1.570796, 1.841951],accel_mss,speed_ms,0,blend_radius_m)
    movel([0.270522, -1.196358, -2.679468, -0.836563, 1.570796, 1.841318],accel_mss,speed_ms,0,blend_radius_m)
    movel([0.270431, -1.195078, -2.680071, -0.837240, 1.570796, 1.841227],accel_mss,speed_ms,0,blend_radius_m)
    movel([0.270763, -1.193575, -2.680777, -0.838038, 1.570796, 1.841559],accel_mss,speed_ms,0,blend_radius_m)
    movel([0.271556, -1.191733, -2.681638, -0.839018, 1.570796, 1.842352],accel_mss,speed_ms,0,blend_radius_m)
    movel([0.273643, -1.188146, -2.683305, -0.840938, 1.570796, 1.844439],accel_mss,speed_ms,0,blend_radius_m)
    movel([0.274008, -1.187409, -2.683646, -0.841334, 1.570796, 1.844804],accel_mss,speed_ms,0,blend_radius_m)
    movel([0.274092, -1.186994, -2.683838, -0.841557, 1.570796, 1.844889],accel_mss,speed_ms,0,blend_radius_m)
    movel([0.273936, -1.186810, -2.683922, -0.841656, 1.570796, 1.844732],accel_mss,speed_ms,0,blend_radius_m)
    movel([0.273577, -1.186895, -2.683883, -0.841611, 1.570796, 1.844373],accel_mss,speed_ms,0,blend_radius_m)
    movel([0.273190, -1.187212, -2.683737, -0.841440, 1.570796, 1.843987],accel_mss,speed_ms,0,blend_radius_m)
    movel([0.271815, -1.189228, -2.682804, -0.840357, 1.570796, 1.842611],accel_mss,speed_ms,0,blend_radius_m)
    movel([0.270634, -1.191251, -2.681863, -0.839275, 1.570796, 1.841430],accel_mss,speed_ms,0,blend_radius_m)
    movel([0.269823, -1.192945, -2.681072, -0.838372, 1.570796, 1.840619],accel_mss,speed_ms,0,blend_radius_m)
    movel([0.269336, -1.194401, -2.680389, -0.837599, 1.570796, 1.840133],accel_mss,speed_ms,0,blend_radius_m)
    movel([0.269115, -1.196218, -2.679534, -0.836637, 1.570796, 1.839911],accel_mss,speed_ms,0,blend_radius_m)
    movel([0.269051, -1.196652, -2.679329, -0.836407, 1.570796, 1.839848],accel_mss,speed_ms,0,blend_radius_m)
    movel([0.268866, -1.197118, -2.679109, -0.836162, 1.570796, 1.839663],accel_mss,speed_ms,0,blend_radius_m)
    movel([0.268459, -1.197542, -2.678909, -0.835938, 1.570796, 1.839256],accel_mss,speed_ms,0,blend_radius_m)
    movel([0.267240, -1.199633, -2.677917, -0.834838, 1.570796, 1.838037],accel_mss,speed_ms,0,blend_radius_m)
    movel([0.266758, -1.200707, -2.677406, -0.834276, 1.570796, 1.837554],accel_mss,speed_ms,0,blend_radius_m)
    movel([0.266120, -1.202821, -2.676396, -0.833171, 1.570796, 1.836916],accel_mss,speed_ms,0,blend_radius_m)
    movel([0.266005, -1.203456, -2.676092, -0.832841, 1.570796, 1.836801],accel_mss,speed_ms,0,blend_radius_m)
    movel([0.265960, -1.205101, -2.675302, -0.831986, 1.570796, 1.836756],accel_mss,speed_ms,0,blend_radius_m)
    movel([0.266285, -1.206688, -2.674536, -0.831164, 1.570796, 1.837082],accel_mss,speed_ms,0,blend_radius_m)
    movel([0.266847, -1.207874, -2.673963, -0.830552, 1.570796, 1.837643],accel_mss,speed_ms,0,blend_radius_m)
    movel([0.267118, -1.208076, -2.673865, -0.830448, 1.570796, 1.837914],accel_mss,speed_ms,0,blend_radius_m)
    movel([0.267528, -1.208074, -2.673866, -0.830449, 1.570796, 1.838324],accel_mss,speed_ms,0,blend_radius_m)
    movel([0.267938, -1.207861, -2.673969, -0.830559, 1.570796, 1.838734],accel_mss,speed_ms,0,blend_radius_m)
    movel([0.268159, -1.207525, -2.674132, -0.830732, 1.570796, 1.838955],accel_mss,speed_ms,0,blend_radius_m)
    movel([0.268142, -1.207040, -2.674366, -0.830982, 1.570796, 1.838938],accel_mss,speed_ms,0,blend_radius_m)
    movel([0.267861, -1.206410, -2.674671, -0.831308, 1.570796, 1.838657],accel_mss,speed_ms,0,blend_radius_m)
    movel([0.267663, -1.205994, -2.674871, -0.831523, 1.570796, 1.838459],accel_mss,speed_ms,0,blend_radius_m)
    movel([0.267238, -1.204511, -2.675585, -0.832292, 1.570796, 1.838034],accel_mss,speed_ms,0,blend_radius_m)
    movel([0.267245, -1.203375, -2.676131, -0.832883, 1.570796, 1.838042],accel_mss,speed_ms,0,blend_radius_m)
    movel([0.267527, -1.201933, -2.676821, -0.833635, 1.570796, 1.838323],accel_mss,speed_ms,0,blend_radius_m)
    movel([0.268014, -1.200429, -2.677539, -0.834421, 1.570796, 1.838810],accel_mss,speed_ms,0,blend_radius_m)
    movel([0.269339, -1.197895, -2.678742, -0.835752, 1.570796, 1.840136],accel_mss,speed_ms,0,blend_radius_m)
    movel([0.269878, -1.198462, -2.678473, -0.835454, 1.570796, 1.840674],accel_mss,speed_ms,0,blend_radius_m)
    movel([0.270786, -1.199008, -2.678214, -0.835167, 1.570796, 1.841582],accel_mss,speed_ms,0,blend_radius_m)
    movel([0.271250, -1.199028, -2.678205, -0.835156, 1.570796, 1.842046],accel_mss,speed_ms,0,blend_radius_m)
    movel([0.271645, -1.198861, -2.678284, -0.835244, 1.570796, 1.842441],accel_mss,speed_ms,0,blend_radius_m)
    movel([0.272020, -1.198260, -2.678569, -0.835560, 1.570796, 1.842817],accel_mss,speed_ms,0,blend_radius_m)
    movel([0.272063, -1.197955, -2.678713, -0.835721, 1.570796, 1.842860],accel_mss,speed_ms,0,blend_radius_m)
    movel([0.271607, -1.197834, -2.678770, -0.835784, 1.570796, 1.842404],accel_mss,speed_ms,0,blend_radius_m)
    movel([0.271155, -1.197426, -2.678964, -0.835999, 1.570796, 1.841951],accel_mss,speed_ms,0,blend_radius_m)
    movel([0.270883, -1.196965, -2.679182, -0.836242, 1.570796, 1.841680],accel_mss,speed_ms,0,blend_radius_m)
    speed_ms = 0.005
    movel([0.270883, -1.187280, -2.674354, -0.850754, 1.570796, 1.841680],accel_mss,speed_ms,0,blend_radius_m)
    speed_ms = 0.040
    movel([0.255364, -1.189309, -2.673406, -0.849674, 1.570796, 1.826160],accel_mss,speed_ms,0,blend_radius_m)
    speed_ms = 0.005
    movel([0.255364, -1.198987, -2.678224, -0.835178, 1.570796, 1.826160],accel_mss,speed_ms,0,blend_radius_m)
    speed_ms = 0.025
    movel([0.255678, -1.198694, -2.678363, -0.835332, 1.570796, 1.826474],accel_mss,speed_ms,0,blend_radius_m)
    movel([0.255840, -1.198369, -2.678517, -0.835503, 1.570796, 1.826636],accel_mss,speed_ms,0,blend_radius_m)
    movel([0.255901, -1.197836, -2.678770, -0.835784, 1.570796, 1.826698],accel_mss,speed_ms,0,blend_radius_m)
    movel([0.255835, -1.192451, -2.681303, -0.838635, 1.570796, 1.826631],accel_mss,speed_ms,0,blend_radius_m)
    movel([0.255666, -1.191484, -2.681754, -0.839151, 1.570796, 1.826462],accel_mss,speed_ms,0,blend_radius_m)
    movel([0.255378, -1.190849, -2.682050, -0.839490, 1.570796, 1.826174],accel_mss,speed_ms,0,blend_radius_m)
    movel([0.254779, -1.190287, -2.682312, -0.839790, 1.570796, 1.825575],accel_mss,speed_ms,0,blend_radius_m)
    movel([0.254012, -1.190021, -2.682435, -0.839932, 1.570796, 1.824808],accel_mss,speed_ms,0,blend_radius_m)
    movel([0.252957, -1.190035, -2.682429, -0.839925, 1.570796, 1.823754],accel_mss,speed_ms,0,blend_radius_m)
    movel([0.251480, -1.190326, -2.682294, -0.839769, 1.570796, 1.822277],accel_mss,speed_ms,0,blend_radius_m)
    movel([0.250086, -1.190717, -2.682112, -0.839560, 1.570796, 1.820882],accel_mss,speed_ms,0,blend_radius_m)
    movel([0.249402, -1.191061, -2.681951, -0.839376, 1.570796, 1.820199],accel_mss,speed_ms,0,blend_radius_m)
    movel([0.249082, -1.191479, -2.681756, -0.839153, 1.570796, 1.819878],accel_mss,speed_ms,0,blend_radius_m)
    movel([0.249025, -1.192044, -2.681493, -0.838852, 1.570796, 1.819821],accel_mss,speed_ms,0,blend_radius_m)
    movel([0.249079, -1.192521, -2.681270, -0.838598, 1.570796, 1.819875],accel_mss,speed_ms,0,blend_radius_m)
    movel([0.248890, -1.192736, -2.681170, -0.838484, 1.570796, 1.819687],accel_mss,speed_ms,0,blend_radius_m)
    movel([0.248360, -1.192798, -2.681141, -0.838451, 1.570796, 1.819156],accel_mss,speed_ms,0,blend_radius_m)
    movel([0.246899, -1.193219, -2.680944, -0.838227, 1.570796, 1.817695],accel_mss,speed_ms,0,blend_radius_m)
    movel([0.246340, -1.193446, -2.680837, -0.838106, 1.570796, 1.817137],accel_mss,speed_ms,0,blend_radius_m)
    movel([0.245053, -1.194140, -2.680512, -0.837737, 1.570796, 1.815849],accel_mss,speed_ms,0,blend_radius_m)
    movel([0.244514, -1.194565, -2.680312, -0.837512, 1.570796, 1.815310],accel_mss,speed_ms,0,blend_radius_m)
    movel([0.243101, -1.196023, -2.679626, -0.836740, 1.570796, 1.813898],accel_mss,speed_ms,0,blend_radius_m)
    movel([0.242544, -1.196830, -2.679245, -0.836313, 1.570796, 1.813340],accel_mss,speed_ms,0,blend_radius_m)
    movel([0.242212, -1.197576, -2.678893, -0.835920, 1.570796, 1.813009],accel_mss,speed_ms,0,blend_radius_m)
    movel([0.242100, -1.198261, -2.678568, -0.835559, 1.570796, 1.812897],accel_mss,speed_ms,0,blend_radius_m)
    movel([0.242223, -1.198598, -2.678409, -0.835382, 1.570796, 1.813019],accel_mss,speed_ms,0,blend_radius_m)
    movel([0.242382, -1.198641, -2.678388, -0.835360, 1.570796, 1.813178],accel_mss,speed_ms,0,blend_radius_m)
    movel([0.242896, -1.198509, -2.678451, -0.835429, 1.570796, 1.813693],accel_mss,speed_ms,0,blend_radius_m)
    movel([0.243071, -1.198378, -2.678513, -0.835498, 1.570796, 1.813867],accel_mss,speed_ms,0,blend_radius_m)
    movel([0.243534, -1.197180, -2.679080, -0.836129, 1.570796, 1.814330],accel_mss,speed_ms,0,blend_radius_m)
    movel([0.243903, -1.196534, -2.679385, -0.836470, 1.570796, 1.814700],accel_mss,speed_ms,0,blend_radius_m)
    movel([0.244382, -1.195943, -2.679664, -0.836782, 1.570796, 1.815178],accel_mss,speed_ms,0,blend_radius_m)
    movel([0.244955, -1.195426, -2.679907, -0.837056, 1.570796, 1.815751],accel_mss,speed_ms,0,blend_radius_m)
    movel([0.245688, -1.194932, -2.680140, -0.837317, 1.570796, 1.816484],accel_mss,speed_ms,0,blend_radius_m)
    movel([0.246440, -1.194562, -2.680313, -0.837513, 1.570796, 1.817237],accel_mss,speed_ms,0,blend_radius_m)
    movel([0.248295, -1.193986, -2.680584, -0.837819, 1.570796, 1.819091],accel_mss,speed_ms,0,blend_radius_m)
    movel([0.249941, -1.193635, -2.680748, -0.838005, 1.570796, 1.820737],accel_mss,speed_ms,0,blend_radius_m)
    movel([0.250179, -1.192710, -2.681182, -0.838497, 1.570796, 1.820976],accel_mss,speed_ms,0,blend_radius_m)
    movel([0.250441, -1.192015, -2.681507, -0.838868, 1.570796, 1.821237],accel_mss,speed_ms,0,blend_radius_m)
    movel([0.250810, -1.191610, -2.681695, -0.839083, 1.570796, 1.821606],accel_mss,speed_ms,0,blend_radius_m)
    movel([0.251370, -1.191392, -2.681797, -0.839200, 1.570796, 1.822166],accel_mss,speed_ms,0,blend_radius_m)
    movel([0.252376, -1.191308, -2.681837, -0.839245, 1.570796, 1.823172],accel_mss,speed_ms,0,blend_radius_m)
    movel([0.253611, -1.191472, -2.681760, -0.839157, 1.570796, 1.824407],accel_mss,speed_ms,0,blend_radius_m)
    movel([0.254268, -1.192048, -2.681491, -0.838850, 1.570796, 1.825064],accel_mss,speed_ms,0,blend_radius_m)
    movel([0.254552, -1.193318, -2.680897, -0.838174, 1.570796, 1.825348],accel_mss,speed_ms,0,blend_radius_m)
    movel([0.254588, -1.197275, -2.679035, -0.836079, 1.570796, 1.825384],accel_mss,speed_ms,0,blend_radius_m)
    movel([0.254619, -1.198257, -2.678570, -0.835562, 1.570796, 1.825415],accel_mss,speed_ms,0,blend_radius_m)
    movel([0.254736, -1.199196, -2.678125, -0.835068, 1.570796, 1.825533],accel_mss,speed_ms,0,blend_radius_m)
    movel([0.255364, -1.198987, -2.678224, -0.835178, 1.570796, 1.826160],accel_mss,speed_ms,0,blend_radius_m)
    movel([0.255678, -1.198694, -2.678363, -0.835332, 1.570796, 1.826474],accel_mss,speed_ms,0,blend_radius_m)
    movel([0.255840, -1.198369, -2.678517, -0.835503, 1.570796, 1.826636],accel_mss,speed_ms,0,blend_radius_m)
    movel([0.255901, -1.197836, -2.678770, -0.835784, 1.570796, 1.826698],accel_mss,speed_ms,0,blend_radius_m)
    movel([0.255882, -1.196235, -2.679526, -0.836628, 1.570796, 1.826679],accel_mss,speed_ms,0,blend_radius_m)
    speed_ms = 0.005
    movel([0.255882, -1.186548, -2.674695, -0.851146, 1.570796, 1.826679],accel_mss,speed_ms,0,blend_radius_m)
    speed_ms = 0.040
    movel([0.250854, -1.179920, -2.677758, -0.854712, 1.570796, 1.821651],accel_mss,speed_ms,0,blend_radius_m)
    speed_ms = 0.005
    movel([0.250854, -1.189627, -2.682618, -0.840143, 1.570796, 1.821651],accel_mss,speed_ms,0,blend_radius_m)
    speed_ms = 0.025
    movel([0.251172, -1.189391, -2.682728, -0.840270, 1.570796, 1.821968],accel_mss,speed_ms,0,blend_radius_m)
    movel([0.251351, -1.189062, -2.682881, -0.840446, 1.570796, 1.822147],accel_mss,speed_ms,0,blend_radius_m)
    movel([0.251397, -1.188034, -2.683357, -0.840998, 1.570796, 1.822193],accel_mss,speed_ms,0,blend_radius_m)
    movel([0.250998, -1.186701, -2.683973, -0.841715, 1.570796, 1.821794],accel_mss,speed_ms,0,blend_radius_m)
    movel([0.250169, -1.185263, -2.684635, -0.842491, 1.570796, 1.820965],accel_mss,speed_ms,0,blend_radius_m)
    movel([0.249306, -1.184311, -2.685072, -0.843006, 1.570796, 1.820103],accel_mss,speed_ms,0,blend_radius_m)
    movel([0.248204, -1.183573, -2.685410, -0.843405, 1.570796, 1.819000],accel_mss,speed_ms,0,blend_radius_m)
    movel([0.247051, -1.183150, -2.685604, -0.843635, 1.570796, 1.817847],accel_mss,speed_ms,0,blend_radius_m)
    movel([0.245860, -1.183222, -2.685571, -0.843596, 1.570796, 1.816657],accel_mss,speed_ms,0,blend_radius_m)
    movel([0.245698, -1.183205, -2.685579, -0.843605, 1.570796, 1.816494],accel_mss,speed_ms,0,blend_radius_m)
    movel([0.245602, -1.183016, -2.685665, -0.843707, 1.570796, 1.816398],accel_mss,speed_ms,0,blend_radius_m)
    movel([0.245643, -1.182466, -2.685917, -0.844007, 1.570796, 1.816440],accel_mss,speed_ms,0,blend_radius_m)
    movel([0.245465, -1.182044, -2.686109, -0.844236, 1.570796, 1.816261],accel_mss,speed_ms,0,blend_radius_m)
    movel([0.243475, -1.179779, -2.687140, -0.845470, 1.570796, 1.814271],accel_mss,speed_ms,0,blend_radius_m)
    movel([0.241371, -1.177716, -2.688074, -0.846599, 1.570796, 1.812167],accel_mss,speed_ms,0,blend_radius_m)
    movel([0.240764, -1.177305, -2.688260, -0.846824, 1.570796, 1.811560],accel_mss,speed_ms,0,blend_radius_m)
    movel([0.240028, -1.177060, -2.688370, -0.846959, 1.570796, 1.810825],accel_mss,speed_ms,0,blend_radius_m)
    movel([0.238980, -1.177001, -2.688397, -0.846991, 1.570796, 1.809776],accel_mss,speed_ms,0,blend_radius_m)
    movel([0.237783, -1.177214, -2.688301, -0.846874, 1.570796, 1.808580],accel_mss,speed_ms,0,blend_radius_m)
    movel([0.236602, -1.177662, -2.688098, -0.846628, 1.570796, 1.807399],accel_mss,speed_ms,0,blend_radius_m)
    movel([0.235619, -1.178289, -2.687815, -0.846285, 1.570796, 1.806415],accel_mss,speed_ms,0,blend_radius_m)
    movel([0.234888, -1.178978, -2.687503, -0.845908, 1.570796, 1.805684],accel_mss,speed_ms,0,blend_radius_m)
    movel([0.234231, -1.179803, -2.687129, -0.845457, 1.570796, 1.805027],accel_mss,speed_ms,0,blend_radius_m)
    movel([0.233721, -1.180659, -2.686740, -0.844990, 1.570796, 1.804518],accel_mss,speed_ms,0,blend_radius_m)
    movel([0.233307, -1.181875, -2.686187, -0.844328, 1.570796, 1.804104],accel_mss,speed_ms,0,blend_radius_m)
    movel([0.233167, -1.182084, -2.686091, -0.844214, 1.570796, 1.803964],accel_mss,speed_ms,0,blend_radius_m)
    movel([0.232432, -1.182384, -2.685954, -0.844051, 1.570796, 1.803228],accel_mss,speed_ms,0,blend_radius_m)
    movel([0.231250, -1.182799, -2.685764, -0.843825, 1.570796, 1.802046],accel_mss,speed_ms,0,blend_radius_m)
    movel([0.228358, -1.184237, -2.685106, -0.843046, 1.570796, 1.799155],accel_mss,speed_ms,0,blend_radius_m)
    movel([0.227307, -1.184931, -2.684788, -0.842671, 1.570796, 1.798103],accel_mss,speed_ms,0,blend_radius_m)
    movel([0.225912, -1.186207, -2.684201, -0.841981, 1.570796, 1.796709],accel_mss,speed_ms,0,blend_radius_m)
    movel([0.225607, -1.186575, -2.684031, -0.841783, 1.570796, 1.796404],accel_mss,speed_ms,0,blend_radius_m)
    movel([0.225013, -1.187628, -2.683545, -0.841216, 1.570796, 1.795809],accel_mss,speed_ms,0,blend_radius_m)
    movel([0.224791, -1.188604, -2.683093, -0.840692, 1.570796, 1.795588],accel_mss,speed_ms,0,blend_radius_m)
    movel([0.225005, -1.189128, -2.682850, -0.840411, 1.570796, 1.795802],accel_mss,speed_ms,0,blend_radius_m)
    movel([0.225242, -1.189186, -2.682823, -0.840380, 1.570796, 1.796038],accel_mss,speed_ms,0,blend_radius_m)
    movel([0.225546, -1.189076, -2.682874, -0.840439, 1.570796, 1.796342],accel_mss,speed_ms,0,blend_radius_m)
    movel([0.225715, -1.188930, -2.682942, -0.840517, 1.570796, 1.796511],accel_mss,speed_ms,0,blend_radius_m)
    movel([0.226101, -1.188030, -2.683359, -0.841000, 1.570796, 1.796897],accel_mss,speed_ms,0,blend_radius_m)
    movel([0.226335, -1.187412, -2.683645, -0.841332, 1.570796, 1.797132],accel_mss,speed_ms,0,blend_radius_m)
    movel([0.226734, -1.186803, -2.683926, -0.841660, 1.570796, 1.797530],accel_mss,speed_ms,0,blend_radius_m)
    movel([0.227305, -1.186186, -2.684210, -0.841993, 1.570796, 1.798102],accel_mss,speed_ms,0,blend_radius_m)
    movel([0.228846, -1.185089, -2.684715, -0.842585, 1.570796, 1.799642],accel_mss,speed_ms,0,blend_radius_m)
    movel([0.229757, -1.184637, -2.684922, -0.842829, 1.570796, 1.800553],accel_mss,speed_ms,0,blend_radius_m)
    movel([0.232963, -1.183522, -2.685434, -0.843433, 1.570796, 1.803759],accel_mss,speed_ms,0,blend_radius_m)
    movel([0.233725, -1.183256, -2.685556, -0.843578, 1.570796, 1.804521],accel_mss,speed_ms,0,blend_radius_m)
    movel([0.234552, -1.182875, -2.685730, -0.843784, 1.570796, 1.805348],accel_mss,speed_ms,0,blend_radius_m)
    movel([0.234665, -1.182704, -2.685808, -0.843877, 1.570796, 1.805461],accel_mss,speed_ms,0,blend_radius_m)
    movel([0.234788, -1.181673, -2.686279, -0.844438, 1.570796, 1.805584],accel_mss,speed_ms,0,blend_radius_m)
    movel([0.234792, -1.181166, -2.686509, -0.844713, 1.570796, 1.805588],accel_mss,speed_ms,0,blend_radius_m)
    movel([0.234969, -1.180481, -2.686821, -0.845087, 1.570796, 1.805766],accel_mss,speed_ms,0,blend_radius_m)
    movel([0.235177, -1.180126, -2.686982, -0.845280, 1.570796, 1.805973],accel_mss,speed_ms,0,blend_radius_m)
    movel([0.235988, -1.179259, -2.687376, -0.845754, 1.570796, 1.806785],accel_mss,speed_ms,0,blend_radius_m)
    movel([0.237028, -1.178635, -2.687658, -0.846095, 1.570796, 1.807825],accel_mss,speed_ms,0,blend_radius_m)
    movel([0.238162, -1.178342, -2.687791, -0.846256, 1.570796, 1.808958],accel_mss,speed_ms,0,blend_radius_m)
    movel([0.239232, -1.178426, -2.687753, -0.846210, 1.570796, 1.810028],accel_mss,speed_ms,0,blend_radius_m)
    movel([0.239970, -1.178788, -2.687590, -0.846012, 1.570796, 1.810766],accel_mss,speed_ms,0,blend_radius_m)
    movel([0.241074, -1.179730, -2.687162, -0.845497, 1.570796, 1.811871],accel_mss,speed_ms,0,blend_radius_m)
    movel([0.243502, -1.182390, -2.685951, -0.844048, 1.570796, 1.814298],accel_mss,speed_ms,0,blend_radius_m)
    movel([0.244468, -1.183618, -2.685390, -0.843381, 1.570796, 1.815264],accel_mss,speed_ms,0,blend_radius_m)
    movel([0.243189, -1.184860, -2.684820, -0.842709, 1.570796, 1.813985],accel_mss,speed_ms,0,blend_radius_m)
    movel([0.242893, -1.185251, -2.684640, -0.842497, 1.570796, 1.813689],accel_mss,speed_ms,0,blend_radius_m)
    movel([0.242130, -1.186343, -2.684138, -0.841908, 1.570796, 1.812926],accel_mss,speed_ms,0,blend_radius_m)
    movel([0.241802, -1.186563, -2.684036, -0.841789, 1.570796, 1.812599],accel_mss,speed_ms,0,blend_radius_m)
    movel([0.240309, -1.187277, -2.683707, -0.841405, 1.570796, 1.811106],accel_mss,speed_ms,0,blend_radius_m)
    movel([0.239374, -1.187874, -2.683431, -0.841084, 1.570796, 1.810170],accel_mss,speed_ms,0,blend_radius_m)
    movel([0.238469, -1.188605, -2.683093, -0.840691, 1.570796, 1.809265],accel_mss,speed_ms,0,blend_radius_m)
    movel([0.237583, -1.189475, -2.682689, -0.840225, 1.570796, 1.808379],accel_mss,speed_ms,0,blend_radius_m)
    movel([0.236683, -1.190567, -2.682181, -0.839640, 1.570796, 1.807479],accel_mss,speed_ms,0,blend_radius_m)
    movel([0.236131, -1.191540, -2.681728, -0.839121, 1.570796, 1.806927],accel_mss,speed_ms,0,blend_radius_m)
    movel([0.236039, -1.192175, -2.681432, -0.838782, 1.570796, 1.806835],accel_mss,speed_ms,0,blend_radius_m)
    movel([0.236150, -1.192351, -2.681350, -0.838689, 1.570796, 1.806946],accel_mss,speed_ms,0,blend_radius_m)
    movel([0.236565, -1.192333, -2.681358, -0.838698, 1.570796, 1.807361],accel_mss,speed_ms,0,blend_radius_m)
    movel([0.236769, -1.192177, -2.681431, -0.838781, 1.570796, 1.807565],accel_mss,speed_ms,0,blend_radius_m)
    movel([0.237233, -1.191542, -2.681727, -0.839120, 1.570796, 1.808029],accel_mss,speed_ms,0,blend_radius_m)
    movel([0.238258, -1.190150, -2.682375, -0.839863, 1.570796, 1.809054],accel_mss,speed_ms,0,blend_radius_m)
    movel([0.239519, -1.188968, -2.682925, -0.840497, 1.570796, 1.810315],accel_mss,speed_ms,0,blend_radius_m)
    movel([0.240856, -1.188132, -2.683312, -0.840945, 1.570796, 1.811653],accel_mss,speed_ms,0,blend_radius_m)
    movel([0.242104, -1.187757, -2.683485, -0.841147, 1.570796, 1.812900],accel_mss,speed_ms,0,blend_radius_m)
    movel([0.242798, -1.187625, -2.683546, -0.841218, 1.570796, 1.813594],accel_mss,speed_ms,0,blend_radius_m)
    movel([0.243221, -1.187389, -2.683655, -0.841345, 1.570796, 1.814017],accel_mss,speed_ms,0,blend_radius_m)
    movel([0.243497, -1.187004, -2.683833, -0.841552, 1.570796, 1.814294],accel_mss,speed_ms,0,blend_radius_m)
    movel([0.243940, -1.185606, -2.684477, -0.842306, 1.570796, 1.814736],accel_mss,speed_ms,0,blend_radius_m)
    movel([0.244169, -1.185310, -2.684614, -0.842466, 1.570796, 1.814965],accel_mss,speed_ms,0,blend_radius_m)
    movel([0.244990, -1.184601, -2.684939, -0.842849, 1.570796, 1.815786],accel_mss,speed_ms,0,blend_radius_m)
    movel([0.245274, -1.184455, -2.685006, -0.842928, 1.570796, 1.816070],accel_mss,speed_ms,0,blend_radius_m)
    movel([0.246177, -1.184480, -2.684995, -0.842914, 1.570796, 1.816973],accel_mss,speed_ms,0,blend_radius_m)
    movel([0.247190, -1.184842, -2.684828, -0.842719, 1.570796, 1.817986],accel_mss,speed_ms,0,blend_radius_m)
    movel([0.248262, -1.185719, -2.684425, -0.842245, 1.570796, 1.819058],accel_mss,speed_ms,0,blend_radius_m)
    movel([0.249220, -1.186908, -2.683877, -0.841604, 1.570796, 1.820016],accel_mss,speed_ms,0,blend_radius_m)
    movel([0.250436, -1.189369, -2.682739, -0.840282, 1.570796, 1.821232],accel_mss,speed_ms,0,blend_radius_m)
    movel([0.250659, -1.189620, -2.682622, -0.840147, 1.570796, 1.821456],accel_mss,speed_ms,0,blend_radius_m)
    movel([0.250854, -1.189627, -2.682618, -0.840143, 1.570796, 1.821651],accel_mss,speed_ms,0,blend_radius_m)
    movel([0.251172, -1.189391, -2.682728, -0.840270, 1.570796, 1.821968],accel_mss,speed_ms,0,blend_radius_m)
    movel([0.251351, -1.189062, -2.682881, -0.840446, 1.570796, 1.822147],accel_mss,speed_ms,0,blend_radius_m)
    movel([0.251397, -1.188034, -2.683357, -0.840998, 1.570796, 1.822193],accel_mss,speed_ms,0,blend_radius_m)
    movel([0.251098, -1.187042, -2.683815, -0.841531, 1.570796, 1.821895],accel_mss,speed_ms,0,blend_radius_m)
    speed_ms = 0.005
    movel([0.251098, -1.177326, -2.678943, -0.856120, 1.570796, 1.821895],accel_mss,speed_ms,0,blend_radius_m)
    speed_ms = 0.040
    movel([0.286619, -1.175258, -2.679883, -0.857247, 1.570796, 1.857415],accel_mss,speed_ms,0,blend_radius_m)
    speed_ms = 0.005
    movel([0.286619, -1.184980, -2.684765, -0.842644, 1.570796, 1.857415],accel_mss,speed_ms,0,blend_radius_m)
    speed_ms = 0.025
    movel([0.286888, -1.184698, -2.684895, -0.842796, 1.570796, 1.857685],accel_mss,speed_ms,0,blend_radius_m)
    movel([0.287131, -1.184139, -2.685151, -0.843099, 1.570796, 1.857927],accel_mss,speed_ms,0,blend_radius_m)
    movel([0.287047, -1.183997, -2.685216, -0.843176, 1.570796, 1.857843],accel_mss,speed_ms,0,blend_radius_m)
    movel([0.285131, -1.183987, -2.685221, -0.843181, 1.570796, 1.855927],accel_mss,speed_ms,0,blend_radius_m)
    movel([0.284397, -1.183801, -2.685306, -0.843282, 1.570796, 1.855193],accel_mss,speed_ms,0,blend_radius_m)
    movel([0.283820, -1.183462, -2.685461, -0.843466, 1.570796, 1.854616],accel_mss,speed_ms,0,blend_radius_m)
    movel([0.283401, -1.182958, -2.685692, -0.843739, 1.570796, 1.854198],accel_mss,speed_ms,0,blend_radius_m)
    movel([0.283198, -1.182378, -2.685957, -0.844054, 1.570796, 1.853994],accel_mss,speed_ms,0,blend_radius_m)
    movel([0.283190, -1.181681, -2.686275, -0.844433, 1.570796, 1.853986],accel_mss,speed_ms,0,blend_radius_m)
    movel([0.283388, -1.180979, -2.686595, -0.844815, 1.570796, 1.854185],accel_mss,speed_ms,0,blend_radius_m)
    movel([0.283803, -1.180261, -2.686921, -0.845207, 1.570796, 1.854599],accel_mss,speed_ms,0,blend_radius_m)
    movel([0.284097, -1.179507, -2.687264, -0.845619, 1.570796, 1.854893],accel_mss,speed_ms,0,blend_radius_m)
    movel([0.284020, -1.179269, -2.687371, -0.845748, 1.570796, 1.854816],accel_mss,speed_ms,0,blend_radius_m)
    movel([0.283537, -1.179119, -2.687439, -0.845830, 1.570796, 1.854333],accel_mss,speed_ms,0,blend_radius_m)
    movel([0.283308, -1.178461, -2.687737, -0.846191, 1.570796, 1.854105],accel_mss,speed_ms,0,blend_radius_m)
    movel([0.283133, -1.176565, -2.688593, -0.847230, 1.570796, 1.853929],accel_mss,speed_ms,0,blend_radius_m)
    movel([0.283249, -1.175411, -2.689113, -0.847866, 1.570796, 1.854045],accel_mss,speed_ms,0,blend_radius_m)
    movel([0.283954, -1.172938, -2.690220, -0.849231, 1.570796, 1.854751],accel_mss,speed_ms,0,blend_radius_m)
    movel([0.284534, -1.171660, -2.690790, -0.849939, 1.570796, 1.855330],accel_mss,speed_ms,0,blend_radius_m)
    movel([0.286108, -1.169102, -2.691926, -0.851361, 1.570796, 1.856905],accel_mss,speed_ms,0,blend_radius_m)
    movel([0.287085, -1.167859, -2.692475, -0.852054, 1.570796, 1.857881],accel_mss,speed_ms,0,blend_radius_m)
    movel([0.288923, -1.165863, -2.693354, -0.853171, 1.570796, 1.859719],accel_mss,speed_ms,0,blend_radius_m)
    movel([0.289212, -1.165437, -2.693541, -0.853410, 1.570796, 1.860008],accel_mss,speed_ms,0,blend_radius_m)
    movel([0.289229, -1.165158, -2.693664, -0.853567, 1.570796, 1.860026],accel_mss,speed_ms,0,blend_radius_m)
    movel([0.288991, -1.164941, -2.693759, -0.853689, 1.570796, 1.859788],accel_mss,speed_ms,0,blend_radius_m)
    movel([0.288746, -1.164927, -2.693765, -0.853697, 1.570796, 1.859543],accel_mss,speed_ms,0,blend_radius_m)
    movel([0.288455, -1.165081, -2.693698, -0.853610, 1.570796, 1.859252],accel_mss,speed_ms,0,blend_radius_m)
    movel([0.287437, -1.165989, -2.693299, -0.853101, 1.570796, 1.858234],accel_mss,speed_ms,0,blend_radius_m)
    movel([0.286224, -1.167338, -2.692705, -0.852345, 1.570796, 1.857020],accel_mss,speed_ms,0,blend_radius_m)
    movel([0.285012, -1.168950, -2.691993, -0.851446, 1.570796, 1.855809],accel_mss,speed_ms,0,blend_radius_m)
    movel([0.283819, -1.170819, -2.691165, -0.850406, 1.570796, 1.854615],accel_mss,speed_ms,0,blend_radius_m)
    movel([0.282921, -1.172578, -2.690381, -0.849430, 1.570796, 1.853718],accel_mss,speed_ms,0,blend_radius_m)
    movel([0.282300, -1.174282, -2.689619, -0.848488, 1.570796, 1.853096],accel_mss,speed_ms,0,blend_radius_m)
    movel([0.281922, -1.175986, -2.688854, -0.847549, 1.570796, 1.852719],accel_mss,speed_ms,0,blend_radius_m)
    movel([0.281810, -1.177316, -2.688255, -0.846818, 1.570796, 1.852606],accel_mss,speed_ms,0,blend_radius_m)
    movel([0.281869, -1.178652, -2.687651, -0.846086, 1.570796, 1.852665],accel_mss,speed_ms,0,blend_radius_m)
    movel([0.282044, -1.179763, -2.687147, -0.845479, 1.570796, 1.852840],accel_mss,speed_ms,0,blend_radius_m)
    movel([0.282451, -1.180138, -2.686977, -0.845274, 1.570796, 1.853247],accel_mss,speed_ms,0,blend_radius_m)
    movel([0.282464, -1.180320, -2.686894, -0.845174, 1.570796, 1.853260],accel_mss,speed_ms,0,blend_radius_m)
    movel([0.281904, -1.182146, -2.686063, -0.844180, 1.570796, 1.852701],accel_mss,speed_ms,0,blend_radius_m)
    movel([0.281872, -1.183086, -2.685633, -0.843670, 1.570796, 1.852669],accel_mss,speed_ms,0,blend_radius_m)
    movel([0.282108, -1.183902, -2.685260, -0.843227, 1.570796, 1.852905],accel_mss,speed_ms,0,blend_radius_m)
    movel([0.282593, -1.184554, -2.684961, -0.842874, 1.570796, 1.853389],accel_mss,speed_ms,0,blend_radius_m)
    movel([0.283618, -1.185190, -2.684669, -0.842530, 1.570796, 1.854415],accel_mss,speed_ms,0,blend_radius_m)
    movel([0.284266, -1.185300, -2.684618, -0.842471, 1.570796, 1.855062],accel_mss,speed_ms,0,blend_radius_m)
    movel([0.285735, -1.185305, -2.684616, -0.842468, 1.570796, 1.856532],accel_mss,speed_ms,0,blend_radius_m)
    movel([0.286093, -1.185248, -2.684642, -0.842499, 1.570796, 1.856889],accel_mss,speed_ms,0,blend_radius_m)
    movel([0.286619, -1.184980, -2.684765, -0.842644, 1.570796, 1.857415],accel_mss,speed_ms,0,blend_radius_m)
    movel([0.286888, -1.184698, -2.684895, -0.842796, 1.570796, 1.857685],accel_mss,speed_ms,0,blend_radius_m)
    movel([0.287131, -1.184139, -2.685151, -0.843099, 1.570796, 1.857927],accel_mss,speed_ms,0,blend_radius_m)
    movel([0.287047, -1.183997, -2.685216, -0.843176, 1.570796, 1.857843],accel_mss,speed_ms,0,blend_radius_m)
    movel([0.285248, -1.183986, -2.685221, -0.843182, 1.570796, 1.856044],accel_mss,speed_ms,0,blend_radius_m)
    speed_ms = 0.005
    movel([0.285248, -1.174261, -2.680335, -0.857793, 1.570796, 1.856044],accel_mss,speed_ms,0,blend_radius_m)
    speed_ms = 0.040
    movel([0.315314, -1.140804, -2.694900, -0.876685, 1.570796, 1.886110],accel_mss,speed_ms,0,blend_radius_m)
    speed_ms = 0.005
    movel([0.315314, -1.150611, -2.699936, -0.861843, 1.570796, 1.886110],accel_mss,speed_ms,0,blend_radius_m)
    speed_ms = 0.025
    movel([0.314615, -1.150672, -2.699910, -0.861807, 1.570796, 1.885411],accel_mss,speed_ms,0,blend_radius_m)
    movel([0.314030, -1.150638, -2.699924, -0.861827, 1.570796, 1.884826],accel_mss,speed_ms,0,blend_radius_m)
    movel([0.311693, -1.150473, -2.699994, -0.861922, 1.570796, 1.882489],accel_mss,speed_ms,0,blend_radius_m)
    movel([0.309738, -1.150673, -2.699909, -0.861807, 1.570796, 1.880534],accel_mss,speed_ms,0,blend_radius_m)
    movel([0.307713, -1.151133, -2.699714, -0.861542, 1.570796, 1.878509],accel_mss,speed_ms,0,blend_radius_m)
    movel([0.305786, -1.151819, -2.699423, -0.861147, 1.570796, 1.876582],accel_mss,speed_ms,0,blend_radius_m)
    movel([0.303092, -1.153186, -2.698841, -0.860362, 1.570796, 1.873888],accel_mss,speed_ms,0,blend_radius_m)
    movel([0.300320, -1.155004, -2.698064, -0.859321, 1.570796, 1.871116],accel_mss,speed_ms,0,blend_radius_m)
    movel([0.297716, -1.157102, -2.697163, -0.858123, 1.570796, 1.868512],accel_mss,speed_ms,0,blend_radius_m)
    movel([0.295514, -1.159300, -2.696215, -0.856874, 1.570796, 1.866310],accel_mss,speed_ms,0,blend_radius_m)
    movel([0.294232, -1.160879, -2.695531, -0.855979, 1.570796, 1.865028],accel_mss,speed_ms,0,blend_radius_m)
    movel([0.293549, -1.162093, -2.695003, -0.855293, 1.570796, 1.864346],accel_mss,speed_ms,0,blend_radius_m)
    movel([0.293356, -1.163124, -2.694554, -0.854711, 1.570796, 1.864153],accel_mss,speed_ms,0,blend_radius_m)
    movel([0.293601, -1.164123, -2.694117, -0.854149, 1.570796, 1.864397],accel_mss,speed_ms,0,blend_radius_m)
    movel([0.293780, -1.164753, -2.693841, -0.853795, 1.570796, 1.864576],accel_mss,speed_ms,0,blend_radius_m)
    movel([0.293763, -1.165466, -2.693529, -0.853394, 1.570796, 1.864560],accel_mss,speed_ms,0,blend_radius_m)
    movel([0.293570, -1.166121, -2.693241, -0.853027, 1.570796, 1.864367],accel_mss,speed_ms,0,blend_radius_m)
    movel([0.293220, -1.166587, -2.693036, -0.852766, 1.570796, 1.864016],accel_mss,speed_ms,0,blend_radius_m)
    movel([0.292642, -1.167187, -2.692772, -0.852430, 1.570796, 1.863438],accel_mss,speed_ms,0,blend_radius_m)
    movel([0.292135, -1.167909, -2.692454, -0.852027, 1.570796, 1.862932],accel_mss,speed_ms,0,blend_radius_m)
    movel([0.291374, -1.169709, -2.691657, -0.851023, 1.570796, 1.862170],accel_mss,speed_ms,0,blend_radius_m)
    movel([0.291099, -1.170961, -2.691101, -0.850327, 1.570796, 1.861895],accel_mss,speed_ms,0,blend_radius_m)
    movel([0.291056, -1.172041, -2.690621, -0.849728, 1.570796, 1.861852],accel_mss,speed_ms,0,blend_radius_m)
    movel([0.291248, -1.172980, -2.690201, -0.849207, 1.570796, 1.862045],accel_mss,speed_ms,0,blend_radius_m)
    movel([0.292278, -1.174667, -2.689447, -0.848276, 1.570796, 1.863075],accel_mss,speed_ms,0,blend_radius_m)
    movel([0.291718, -1.176581, -2.688586, -0.847222, 1.570796, 1.862514],accel_mss,speed_ms,0,blend_radius_m)
    movel([0.291364, -1.178095, -2.687903, -0.846391, 1.570796, 1.862160],accel_mss,speed_ms,0,blend_radius_m)
    movel([0.291302, -1.179246, -2.687382, -0.845761, 1.570796, 1.862098],accel_mss,speed_ms,0,blend_radius_m)
    movel([0.291534, -1.180211, -2.686944, -0.845234, 1.570796, 1.862330],accel_mss,speed_ms,0,blend_radius_m)
    movel([0.292084, -1.181146, -2.686519, -0.844725, 1.570796, 1.862881],accel_mss,speed_ms,0,blend_radius_m)
    movel([0.292452, -1.181723, -2.686256, -0.844410, 1.570796, 1.863248],accel_mss,speed_ms,0,blend_radius_m)
    movel([0.292557, -1.182195, -2.686040, -0.844154, 1.570796, 1.863353],accel_mss,speed_ms,0,blend_radius_m)
    movel([0.292420, -1.182572, -2.685868, -0.843948, 1.570796, 1.863216],accel_mss,speed_ms,0,blend_radius_m)
    movel([0.292084, -1.182881, -2.685727, -0.843781, 1.570796, 1.862880],accel_mss,speed_ms,0,blend_radius_m)
    movel([0.291599, -1.182907, -2.685715, -0.843767, 1.570796, 1.862395],accel_mss,speed_ms,0,blend_radius_m)
    movel([0.290967, -1.182262, -2.686010, -0.844117, 1.570796, 1.861763],accel_mss,speed_ms,0,blend_radius_m)
    movel([0.290399, -1.181349, -2.686426, -0.844614, 1.570796, 1.861195],accel_mss,speed_ms,0,blend_radius_m)
    movel([0.290052, -1.180315, -2.686897, -0.845177, 1.570796, 1.860849],accel_mss,speed_ms,0,blend_radius_m)
    movel([0.289921, -1.178962, -2.687510, -0.845916, 1.570796, 1.860717],accel_mss,speed_ms,0,blend_radius_m)
    movel([0.290018, -1.178289, -2.687815, -0.846285, 1.570796, 1.860815],accel_mss,speed_ms,0,blend_radius_m)
    movel([0.290598, -1.175773, -2.688950, -0.847666, 1.570796, 1.861395],accel_mss,speed_ms,0,blend_radius_m)
    movel([0.290557, -1.175356, -2.689137, -0.847896, 1.570796, 1.861354],accel_mss,speed_ms,0,blend_radius_m)
    movel([0.289995, -1.174027, -2.689733, -0.848629, 1.570796, 1.860791],accel_mss,speed_ms,0,blend_radius_m)
    movel([0.289750, -1.173019, -2.690184, -0.849186, 1.570796, 1.860546],accel_mss,speed_ms,0,blend_radius_m)
    movel([0.289679, -1.171982, -2.690647, -0.849760, 1.570796, 1.860475],accel_mss,speed_ms,0,blend_radius_m)
    movel([0.289783, -1.170857, -2.691148, -0.850385, 1.570796, 1.860579],accel_mss,speed_ms,0,blend_radius_m)
    movel([0.290038, -1.169795, -2.691619, -0.850975, 1.570796, 1.860835],accel_mss,speed_ms,0,blend_radius_m)
    movel([0.290466, -1.168697, -2.692105, -0.851587, 1.570796, 1.861262],accel_mss,speed_ms,0,blend_radius_m)
    movel([0.291014, -1.167717, -2.692538, -0.852134, 1.570796, 1.861811],accel_mss,speed_ms,0,blend_radius_m)
    movel([0.291733, -1.166783, -2.692950, -0.852656, 1.570796, 1.862529],accel_mss,speed_ms,0,blend_radius_m)
    movel([0.292496, -1.165923, -2.693328, -0.853138, 1.570796, 1.863292],accel_mss,speed_ms,0,blend_radius_m)
    movel([0.292182, -1.164857, -2.693796, -0.853736, 1.570796, 1.862978],accel_mss,speed_ms,0,blend_radius_m)
    movel([0.292034, -1.163840, -2.694241, -0.854308, 1.570796, 1.862830],accel_mss,speed_ms,0,blend_radius_m)
    movel([0.292166, -1.162774, -2.694706, -0.854908, 1.570796, 1.862963],accel_mss,speed_ms,0,blend_radius_m)
    movel([0.292594, -1.161641, -2.695200, -0.855548, 1.570796, 1.863391],accel_mss,speed_ms,0,blend_radius_m)
    movel([0.293313, -1.160418, -2.695731, -0.856240, 1.570796, 1.864110],accel_mss,speed_ms,0,blend_radius_m)
    movel([0.294423, -1.159056, -2.696321, -0.857012, 1.570796, 1.865219],accel_mss,speed_ms,0,blend_radius_m)
    movel([0.296451, -1.157016, -2.697201, -0.858172, 1.570796, 1.867248],accel_mss,speed_ms,0,blend_radius_m)
    movel([0.298621, -1.155009, -2.698062, -0.859318, 1.570796, 1.869417],accel_mss,speed_ms,0,blend_radius_m)
    movel([0.300305, -1.153670, -2.698634, -0.860084, 1.570796, 1.871101],accel_mss,speed_ms,0,blend_radius_m)
    movel([0.302226, -1.152415, -2.699170, -0.860805, 1.570796, 1.873022],accel_mss,speed_ms,0,blend_radius_m)
    movel([0.304176, -1.151356, -2.699619, -0.861413, 1.570796, 1.874972],accel_mss,speed_ms,0,blend_radius_m)
    movel([0.306205, -1.150461, -2.699999, -0.861929, 1.570796, 1.877001],accel_mss,speed_ms,0,blend_radius_m)
    movel([0.308208, -1.149771, -2.700291, -0.862327, 1.570796, 1.879004],accel_mss,speed_ms,0,blend_radius_m)
    movel([0.310151, -1.149301, -2.700490, -0.862598, 1.570796, 1.880947],accel_mss,speed_ms,0,blend_radius_m)
    movel([0.312023, -1.149055, -2.700594, -0.862740, 1.570796, 1.882819],accel_mss,speed_ms,0,blend_radius_m)
    movel([0.313699, -1.149054, -2.700594, -0.862741, 1.570796, 1.884495],accel_mss,speed_ms,0,blend_radius_m)
    movel([0.315241, -1.149302, -2.700489, -0.862597, 1.570796, 1.886037],accel_mss,speed_ms,0,blend_radius_m)
    movel([0.315653, -1.149518, -2.700398, -0.862473, 1.570796, 1.886449],accel_mss,speed_ms,0,blend_radius_m)
    movel([0.315810, -1.149883, -2.700244, -0.862262, 1.570796, 1.886606],accel_mss,speed_ms,0,blend_radius_m)
    movel([0.315675, -1.150279, -2.700076, -0.862034, 1.570796, 1.886471],accel_mss,speed_ms,0,blend_radius_m)
    movel([0.315314, -1.150611, -2.699936, -0.861843, 1.570796, 1.886110],accel_mss,speed_ms,0,blend_radius_m)
    movel([0.314615, -1.150672, -2.699910, -0.861807, 1.570796, 1.885411],accel_mss,speed_ms,0,blend_radius_m)
    movel([0.314030, -1.150638, -2.699924, -0.861827, 1.570796, 1.884826],accel_mss,speed_ms,0,blend_radius_m)
    movel([0.312501, -1.150532, -2.699969, -0.861888, 1.570796, 1.883297],accel_mss,speed_ms,0,blend_radius_m)
    speed_ms = 0.005
    movel([0.312501, -1.140725, -2.694933, -0.876731, 1.570796, 1.883297],accel_mss,speed_ms,0,blend_radius_m)
    speed_ms = 0.040
    movel([0.330564, -1.150947, -2.690604, -0.870838, 1.570796, 1.901361],accel_mss,speed_ms,0,blend_radius_m)
    speed_ms = 0.005
    movel([0.330564, -1.160732, -2.695595, -0.856062, 1.570796, 1.901361],accel_mss,speed_ms,0,blend_radius_m)
    speed_ms = 0.025
    movel([0.330341, -1.160709, -2.695605, -0.856075, 1.570796, 1.901138],accel_mss,speed_ms,0,blend_radius_m)
    movel([0.329903, -1.160225, -2.695815, -0.856349, 1.570796, 1.900699],accel_mss,speed_ms,0,blend_radius_m)
    movel([0.327422, -1.156688, -2.697342, -0.858359, 1.570796, 1.898218],accel_mss,speed_ms,0,blend_radius_m)
    movel([0.325962, -1.154973, -2.698077, -0.859338, 1.570796, 1.896758],accel_mss,speed_ms,0,blend_radius_m)
    movel([0.324619, -1.153780, -2.698588, -0.860022, 1.570796, 1.895416],accel_mss,speed_ms,0,blend_radius_m)
    movel([0.323055, -1.152831, -2.698992, -0.860565, 1.570796, 1.893851],accel_mss,speed_ms,0,blend_radius_m)
    movel([0.321507, -1.152257, -2.699237, -0.860895, 1.570796, 1.892303],accel_mss,speed_ms,0,blend_radius_m)
    movel([0.319774, -1.151965, -2.699361, -0.861063, 1.570796, 1.890571],accel_mss,speed_ms,0,blend_radius_m)
    movel([0.317908, -1.151964, -2.699361, -0.861064, 1.570796, 1.888704],accel_mss,speed_ms,0,blend_radius_m)
    movel([0.315914, -1.152256, -2.699237, -0.860896, 1.570796, 1.886710],accel_mss,speed_ms,0,blend_radius_m)
    movel([0.313852, -1.152813, -2.699000, -0.860576, 1.570796, 1.884648],accel_mss,speed_ms,0,blend_radius_m)
    movel([0.312994, -1.153164, -2.698850, -0.860374, 1.570796, 1.883791],accel_mss,speed_ms,0,blend_radius_m)
    movel([0.309997, -1.154816, -2.698145, -0.859428, 1.570796, 1.880794],accel_mss,speed_ms,0,blend_radius_m)
    movel([0.308659, -1.155885, -2.697687, -0.858818, 1.570796, 1.879456],accel_mss,speed_ms,0,blend_radius_m)
    movel([0.307739, -1.157048, -2.697187, -0.858154, 1.570796, 1.878535],accel_mss,speed_ms,0,blend_radius_m)
    movel([0.307072, -1.158460, -2.696578, -0.857351, 1.570796, 1.877868],accel_mss,speed_ms,0,blend_radius_m)
    movel([0.306749, -1.159391, -2.696176, -0.856822, 1.570796, 1.877546],accel_mss,speed_ms,0,blend_radius_m)
    movel([0.305275, -1.159870, -2.695969, -0.856551, 1.570796, 1.876072],accel_mss,speed_ms,0,blend_radius_m)
    movel([0.303894, -1.160437, -2.695723, -0.856229, 1.570796, 1.874691],accel_mss,speed_ms,0,blend_radius_m)
    movel([0.302617, -1.161210, -2.695387, -0.855792, 1.570796, 1.873414],accel_mss,speed_ms,0,blend_radius_m)
    movel([0.301445, -1.162187, -2.694962, -0.855240, 1.570796, 1.872242],accel_mss,speed_ms,0,blend_radius_m)
    movel([0.300377, -1.163363, -2.694449, -0.854576, 1.570796, 1.871173],accel_mss,speed_ms,0,blend_radius_m)
    movel([0.299472, -1.164674, -2.693876, -0.853839, 1.570796, 1.870268],accel_mss,speed_ms,0,blend_radius_m)
    movel([0.299212, -1.165270, -2.693615, -0.853504, 1.570796, 1.870008],accel_mss,speed_ms,0,blend_radius_m)
    movel([0.298716, -1.167186, -2.692772, -0.852431, 1.570796, 1.869512],accel_mss,speed_ms,0,blend_radius_m)
    movel([0.298670, -1.168206, -2.692322, -0.851861, 1.570796, 1.869466],accel_mss,speed_ms,0,blend_radius_m)
    movel([0.298783, -1.169018, -2.691963, -0.851408, 1.570796, 1.869580],accel_mss,speed_ms,0,blend_radius_m)
    movel([0.299074, -1.169391, -2.691798, -0.851200, 1.570796, 1.869871],accel_mss,speed_ms,0,blend_radius_m)
    movel([0.299181, -1.169609, -2.691701, -0.851078, 1.570796, 1.869978],accel_mss,speed_ms,0,blend_radius_m)
    movel([0.299059, -1.169979, -2.691538, -0.850873, 1.570796, 1.869855],accel_mss,speed_ms,0,blend_radius_m)
    movel([0.298029, -1.171218, -2.690987, -0.850184, 1.570796, 1.868826],accel_mss,speed_ms,0,blend_radius_m)
    movel([0.297342, -1.171992, -2.690642, -0.849755, 1.570796, 1.868138],accel_mss,speed_ms,0,blend_radius_m)
    movel([0.296221, -1.173730, -2.689866, -0.848793, 1.570796, 1.867017],accel_mss,speed_ms,0,blend_radius_m)
    movel([0.295912, -1.174497, -2.689523, -0.848369, 1.570796, 1.866708],accel_mss,speed_ms,0,blend_radius_m)
    movel([0.295851, -1.176623, -2.688567, -0.847199, 1.570796, 1.866647],accel_mss,speed_ms,0,blend_radius_m)
    movel([0.295881, -1.177717, -2.688074, -0.846598, 1.570796, 1.866678],accel_mss,speed_ms,0,blend_radius_m)
    movel([0.295853, -1.180600, -2.686767, -0.845022, 1.570796, 1.866650],accel_mss,speed_ms,0,blend_radius_m)
    movel([0.295776, -1.180820, -2.686667, -0.844902, 1.570796, 1.866573],accel_mss,speed_ms,0,blend_radius_m)
    movel([0.295324, -1.181183, -2.686502, -0.844704, 1.570796, 1.866120],accel_mss,speed_ms,0,blend_radius_m)
    movel([0.295147, -1.181242, -2.686475, -0.844672, 1.570796, 1.865943],accel_mss,speed_ms,0,blend_radius_m)
    movel([0.294864, -1.181150, -2.686517, -0.844722, 1.570796, 1.865660],accel_mss,speed_ms,0,blend_radius_m)
    movel([0.294694, -1.180670, -2.686735, -0.844984, 1.570796, 1.865490],accel_mss,speed_ms,0,blend_radius_m)
    movel([0.294468, -1.177649, -2.688104, -0.846635, 1.570796, 1.865265],accel_mss,speed_ms,0,blend_radius_m)
    movel([0.294543, -1.175723, -2.688972, -0.847694, 1.570796, 1.865339],accel_mss,speed_ms,0,blend_radius_m)
    movel([0.294956, -1.173994, -2.689748, -0.848647, 1.570796, 1.865752],accel_mss,speed_ms,0,blend_radius_m)
    movel([0.295721, -1.172423, -2.690450, -0.849516, 1.570796, 1.866517],accel_mss,speed_ms,0,blend_radius_m)
    movel([0.296837, -1.170971, -2.691097, -0.850321, 1.570796, 1.867633],accel_mss,speed_ms,0,blend_radius_m)
    movel([0.297554, -1.170204, -2.691438, -0.850748, 1.570796, 1.868351],accel_mss,speed_ms,0,blend_radius_m)
    movel([0.297337, -1.167906, -2.692455, -0.852028, 1.570796, 1.868133],accel_mss,speed_ms,0,blend_radius_m)
    movel([0.297604, -1.166489, -2.693079, -0.852821, 1.570796, 1.868400],accel_mss,speed_ms,0,blend_radius_m)
    movel([0.298106, -1.165037, -2.693717, -0.853635, 1.570796, 1.868903],accel_mss,speed_ms,0,blend_radius_m)
    movel([0.298782, -1.163781, -2.694267, -0.854341, 1.570796, 1.869579],accel_mss,speed_ms,0,blend_radius_m)
    movel([0.300034, -1.162202, -2.694956, -0.855231, 1.570796, 1.870830],accel_mss,speed_ms,0,blend_radius_m)
    movel([0.301657, -1.160695, -2.695611, -0.856083, 1.570796, 1.872454],accel_mss,speed_ms,0,blend_radius_m)
    movel([0.303428, -1.159450, -2.696151, -0.856789, 1.570796, 1.874224],accel_mss,speed_ms,0,blend_radius_m)
    movel([0.305117, -1.158647, -2.696498, -0.857245, 1.570796, 1.875913],accel_mss,speed_ms,0,blend_radius_m)
    movel([0.305966, -1.158277, -2.696657, -0.857454, 1.570796, 1.876763],accel_mss,speed_ms,0,blend_radius_m)
    movel([0.306111, -1.158107, -2.696731, -0.857551, 1.570796, 1.876908],accel_mss,speed_ms,0,blend_radius_m)
    movel([0.306523, -1.156986, -2.697214, -0.858190, 1.570796, 1.877319],accel_mss,speed_ms,0,blend_radius_m)
    movel([0.306747, -1.156613, -2.697374, -0.858402, 1.570796, 1.877544],accel_mss,speed_ms,0,blend_radius_m)
    movel([0.307476, -1.155654, -2.697785, -0.858949, 1.570796, 1.878273],accel_mss,speed_ms,0,blend_radius_m)
    movel([0.308347, -1.154796, -2.698153, -0.859440, 1.570796, 1.879144],accel_mss,speed_ms,0,blend_radius_m)
    movel([0.309487, -1.153902, -2.698535, -0.859951, 1.570796, 1.880283],accel_mss,speed_ms,0,blend_radius_m)
    movel([0.310666, -1.153129, -2.698865, -0.860395, 1.570796, 1.881462],accel_mss,speed_ms,0,blend_radius_m)
    movel([0.312068, -1.152374, -2.699187, -0.860828, 1.570796, 1.882864],accel_mss,speed_ms,0,blend_radius_m)
    movel([0.313470, -1.151766, -2.699446, -0.861178, 1.570796, 1.884266],accel_mss,speed_ms,0,blend_radius_m)
    movel([0.316489, -1.150865, -2.699828, -0.861696, 1.570796, 1.887286],accel_mss,speed_ms,0,blend_radius_m)
    movel([0.318328, -1.150563, -2.699956, -0.861870, 1.570796, 1.889125],accel_mss,speed_ms,0,blend_radius_m)
    movel([0.319922, -1.150503, -2.699981, -0.861905, 1.570796, 1.890719],accel_mss,speed_ms,0,blend_radius_m)
    movel([0.321440, -1.150681, -2.699906, -0.861802, 1.570796, 1.892236],accel_mss,speed_ms,0,blend_radius_m)
    movel([0.323038, -1.151114, -2.699722, -0.861553, 1.570796, 1.893835],accel_mss,speed_ms,0,blend_radius_m)
    movel([0.324964, -1.151992, -2.699349, -0.861048, 1.570796, 1.895760],accel_mss,speed_ms,0,blend_radius_m)
    movel([0.326646, -1.153232, -2.698822, -0.860336, 1.570796, 1.897442],accel_mss,speed_ms,0,blend_radius_m)
    movel([0.328267, -1.155000, -2.698066, -0.859323, 1.570796, 1.899063],accel_mss,speed_ms,0,blend_radius_m)
    movel([0.330866, -1.158912, -2.696383, -0.857094, 1.570796, 1.901662],accel_mss,speed_ms,0,blend_radius_m)
    movel([0.331156, -1.159778, -2.696008, -0.856603, 1.570796, 1.901953],accel_mss,speed_ms,0,blend_radius_m)
    movel([0.331017, -1.160335, -2.695767, -0.856287, 1.570796, 1.901813],accel_mss,speed_ms,0,blend_radius_m)
    movel([0.330564, -1.160732, -2.695595, -0.856062, 1.570796, 1.901361],accel_mss,speed_ms,0,blend_radius_m)
    movel([0.330341, -1.160709, -2.695605, -0.856075, 1.570796, 1.901138],accel_mss,speed_ms,0,blend_radius_m)
    movel([0.329903, -1.160225, -2.695815, -0.856349, 1.570796, 1.900699],accel_mss,speed_ms,0,blend_radius_m)
    movel([0.329043, -1.158994, -2.696348, -0.857047, 1.570796, 1.899840],accel_mss,speed_ms,0,blend_radius_m)
    speed_ms = 0.005
    movel([0.329043, -1.149205, -2.691349, -0.871835, 1.570796, 1.899840],accel_mss,speed_ms,0,blend_radius_m)
    speed_ms = 0.040
    movel([0.331713, -1.158475, -2.687349, -0.866565, 1.570796, 1.902510],accel_mss,speed_ms,0,blend_radius_m)
    speed_ms = 0.005
    movel([0.331713, -1.168242, -2.692306, -0.851841, 1.570796, 1.902510],accel_mss,speed_ms,0,blend_radius_m)
    speed_ms = 0.025
    movel([0.331306, -1.168113, -2.692363, -0.851912, 1.570796, 1.902103],accel_mss,speed_ms,0,blend_radius_m)
    movel([0.331181, -1.167790, -2.692506, -0.852093, 1.570796, 1.901977],accel_mss,speed_ms,0,blend_radius_m)
    movel([0.330488, -1.165082, -2.693697, -0.853610, 1.570796, 1.901285],accel_mss,speed_ms,0,blend_radius_m)
    movel([0.329418, -1.163092, -2.694568, -0.854729, 1.570796, 1.900215],accel_mss,speed_ms,0,blend_radius_m)
    movel([0.327976, -1.161415, -2.695298, -0.855676, 1.570796, 1.898772],accel_mss,speed_ms,0,blend_radius_m)
    movel([0.326286, -1.160232, -2.695812, -0.856345, 1.570796, 1.897083],accel_mss,speed_ms,0,blend_radius_m)
    movel([0.325017, -1.159721, -2.696033, -0.856635, 1.570796, 1.895813],accel_mss,speed_ms,0,blend_radius_m)
    movel([0.323332, -1.159309, -2.696211, -0.856869, 1.570796, 1.894129],accel_mss,speed_ms,0,blend_radius_m)
    movel([0.321666, -1.159053, -2.696322, -0.857014, 1.570796, 1.892462],accel_mss,speed_ms,0,blend_radius_m)
    movel([0.320604, -1.159119, -2.696294, -0.856976, 1.570796, 1.891400],accel_mss,speed_ms,0,blend_radius_m)
    movel([0.319128, -1.159715, -2.696036, -0.856638, 1.570796, 1.889924],accel_mss,speed_ms,0,blend_radius_m)
    movel([0.318351, -1.160251, -2.695804, -0.856335, 1.570796, 1.889148],accel_mss,speed_ms,0,blend_radius_m)
    movel([0.316474, -1.161927, -2.695075, -0.855386, 1.570796, 1.887270],accel_mss,speed_ms,0,blend_radius_m)
    movel([0.313923, -1.162515, -2.694819, -0.855054, 1.570796, 1.884719],accel_mss,speed_ms,0,blend_radius_m)
    movel([0.311493, -1.163182, -2.694529, -0.854679, 1.570796, 1.882289],accel_mss,speed_ms,0,blend_radius_m)
    movel([0.310725, -1.163546, -2.694369, -0.854473, 1.570796, 1.881521],accel_mss,speed_ms,0,blend_radius_m)
    movel([0.308314, -1.165097, -2.693690, -0.853601, 1.570796, 1.879110],accel_mss,speed_ms,0,blend_radius_m)
    movel([0.307457, -1.165878, -2.693348, -0.853163, 1.570796, 1.878254],accel_mss,speed_ms,0,blend_radius_m)
    movel([0.306883, -1.166716, -2.692979, -0.852694, 1.570796, 1.877680],accel_mss,speed_ms,0,blend_radius_m)
    movel([0.306453, -1.167771, -2.692514, -0.852104, 1.570796, 1.877249],accel_mss,speed_ms,0,blend_radius_m)
    movel([0.306245, -1.168703, -2.692103, -0.851583, 1.570796, 1.877041],accel_mss,speed_ms,0,blend_radius_m)
    movel([0.306317, -1.168871, -2.692028, -0.851490, 1.570796, 1.877113],accel_mss,speed_ms,0,blend_radius_m)
    movel([0.306750, -1.169089, -2.691932, -0.851368, 1.570796, 1.877546],accel_mss,speed_ms,0,blend_radius_m)
    movel([0.306794, -1.169237, -2.691866, -0.851286, 1.570796, 1.877590],accel_mss,speed_ms,0,blend_radius_m)
    movel([0.306593, -1.169712, -2.691656, -0.851021, 1.570796, 1.877390],accel_mss,speed_ms,0,blend_radius_m)
    movel([0.306273, -1.169988, -2.691533, -0.850867, 1.570796, 1.877070],accel_mss,speed_ms,0,blend_radius_m)
    movel([0.304136, -1.171018, -2.691076, -0.850295, 1.570796, 1.874933],accel_mss,speed_ms,0,blend_radius_m)
    movel([0.303280, -1.171628, -2.690804, -0.849956, 1.570796, 1.874076],accel_mss,speed_ms,0,blend_radius_m)
    movel([0.301531, -1.173235, -2.690087, -0.849066, 1.570796, 1.872327],accel_mss,speed_ms,0,blend_radius_m)
    movel([0.301020, -1.173828, -2.689822, -0.848738, 1.570796, 1.871816],accel_mss,speed_ms,0,blend_radius_m)
    movel([0.300389, -1.174911, -2.689337, -0.848141, 1.570796, 1.871186],accel_mss,speed_ms,0,blend_radius_m)
    movel([0.300062, -1.175767, -2.688952, -0.847669, 1.570796, 1.870858],accel_mss,speed_ms,0,blend_radius_m)
    movel([0.299607, -1.177615, -2.688120, -0.846654, 1.570796, 1.870404],accel_mss,speed_ms,0,blend_radius_m)
    movel([0.299612, -1.178043, -2.687926, -0.846420, 1.570796, 1.870409],accel_mss,speed_ms,0,blend_radius_m)
    movel([0.299615, -1.178734, -2.687614, -0.846041, 1.570796, 1.870411],accel_mss,speed_ms,0,blend_radius_m)
    movel([0.299503, -1.178945, -2.687518, -0.845926, 1.570796, 1.870299],accel_mss,speed_ms,0,blend_radius_m)
    movel([0.298972, -1.179400, -2.687312, -0.845677, 1.570796, 1.869769],accel_mss,speed_ms,0,blend_radius_m)
    movel([0.298670, -1.179460, -2.687285, -0.845644, 1.570796, 1.869466],accel_mss,speed_ms,0,blend_radius_m)
    movel([0.298302, -1.179128, -2.687435, -0.845825, 1.570796, 1.869098],accel_mss,speed_ms,0,blend_radius_m)
    movel([0.298322, -1.178019, -2.687937, -0.846433, 1.570796, 1.869118],accel_mss,speed_ms,0,blend_radius_m)
    movel([0.299097, -1.175195, -2.689210, -0.847985, 1.570796, 1.869893],accel_mss,speed_ms,0,blend_radius_m)
    movel([0.299377, -1.174512, -2.689516, -0.848361, 1.570796, 1.870173],accel_mss,speed_ms,0,blend_radius_m)
    movel([0.300237, -1.173205, -2.690101, -0.849083, 1.570796, 1.871033],accel_mss,speed_ms,0,blend_radius_m)
    movel([0.301128, -1.172172, -2.690562, -0.849655, 1.570796, 1.871924],accel_mss,speed_ms,0,blend_radius_m)
    movel([0.302132, -1.171214, -2.690989, -0.850186, 1.570796, 1.872929],accel_mss,speed_ms,0,blend_radius_m)
    movel([0.303176, -1.170393, -2.691354, -0.850642, 1.570796, 1.873972],accel_mss,speed_ms,0,blend_radius_m)
    movel([0.304919, -1.169330, -2.691825, -0.851234, 1.570796, 1.875715],accel_mss,speed_ms,0,blend_radius_m)
    movel([0.305106, -1.169138, -2.691910, -0.851341, 1.570796, 1.875903],accel_mss,speed_ms,0,blend_radius_m)
    movel([0.305251, -1.168250, -2.692303, -0.851836, 1.570796, 1.876047],accel_mss,speed_ms,0,blend_radius_m)
    movel([0.305493, -1.167355, -2.692698, -0.852336, 1.570796, 1.876289],accel_mss,speed_ms,0,blend_radius_m)
    movel([0.305832, -1.166483, -2.693082, -0.852824, 1.570796, 1.876628],accel_mss,speed_ms,0,blend_radius_m)
    movel([0.306211, -1.165835, -2.693367, -0.853187, 1.570796, 1.877008],accel_mss,speed_ms,0,blend_radius_m)
    movel([0.306836, -1.165086, -2.693695, -0.853608, 1.570796, 1.877632],accel_mss,speed_ms,0,blend_radius_m)
    movel([0.307551, -1.164418, -2.693988, -0.853983, 1.570796, 1.878347],accel_mss,speed_ms,0,blend_radius_m)
    movel([0.309421, -1.163106, -2.694562, -0.854721, 1.570796, 1.880217],accel_mss,speed_ms,0,blend_radius_m)
    movel([0.311698, -1.161982, -2.695052, -0.855356, 1.570796, 1.882494],accel_mss,speed_ms,0,blend_radius_m)
    movel([0.316256, -1.160519, -2.695688, -0.856183, 1.570796, 1.887052],accel_mss,speed_ms,0,blend_radius_m)
    movel([0.316728, -1.160293, -2.695785, -0.856311, 1.570796, 1.887525],accel_mss,speed_ms,0,blend_radius_m)
    movel([0.317927, -1.159215, -2.696252, -0.856922, 1.570796, 1.888723],accel_mss,speed_ms,0,blend_radius_m)
    movel([0.318329, -1.158914, -2.696382, -0.857093, 1.570796, 1.889125],accel_mss,speed_ms,0,blend_radius_m)
    movel([0.319436, -1.158287, -2.696653, -0.857449, 1.570796, 1.890232],accel_mss,speed_ms,0,blend_radius_m)
    movel([0.320040, -1.158088, -2.696739, -0.857562, 1.570796, 1.890837],accel_mss,speed_ms,0,blend_radius_m)
    movel([0.320882, -1.157898, -2.696821, -0.857670, 1.570796, 1.891679],accel_mss,speed_ms,0,blend_radius_m)
    movel([0.322944, -1.157677, -2.696916, -0.857796, 1.570796, 1.893740],accel_mss,speed_ms,0,blend_radius_m)
    movel([0.324806, -1.157871, -2.696832, -0.857686, 1.570796, 1.895602],accel_mss,speed_ms,0,blend_radius_m)
    movel([0.326669, -1.158486, -2.696567, -0.857336, 1.570796, 1.897466],accel_mss,speed_ms,0,blend_radius_m)
    movel([0.328292, -1.159413, -2.696166, -0.856809, 1.570796, 1.899088],accel_mss,speed_ms,0,blend_radius_m)
    movel([0.329758, -1.160703, -2.695607, -0.856078, 1.570796, 1.900554],accel_mss,speed_ms,0,blend_radius_m)
    movel([0.330942, -1.162270, -2.694926, -0.855193, 1.570796, 1.901738],accel_mss,speed_ms,0,blend_radius_m)
    movel([0.331828, -1.164089, -2.694132, -0.854168, 1.570796, 1.902624],accel_mss,speed_ms,0,blend_radius_m)
    movel([0.332407, -1.166129, -2.693237, -0.853022, 1.570796, 1.903203],accel_mss,speed_ms,0,blend_radius_m)
